// TIA Portal project "PLC_DoAn" (V16)

(* hardware
DEVICE "S71500/ET200MP station_1"  S7-1500 station
   slot 0: "Rail_0"  Rack  6ES7 590-1***0-0AA0
   slot 1: "PLC_1"  CPU 1512C-1 PN  6ES7 512-1CK01-0AB0  V2.8
      slot 3: "CPU display_1"  6ES7591-1AA00-0AA0
      slot 32768: "PROFINET interface_1"  X1
         slot 32769: "Port_1"  X1 P1
         slot 32770: "Port_2"  X1 P2
      slot 34817: "Virtual CP interface port_1"  Virtual CP interface port  Virtual CP interface port
   slot 2: "DQ 16x24VDC/0.5A BA_1"  DQ 16x24VDC/0.5A BA  6ES7 522-1BH10-0AA0  V1.1
DEVICE "PC-System_1"  SIMATIC PC station
   slot 0: "SIMATIC PC station"  Rail  SIMATIC PC-Station  V1.0
      slot 125: "Stationmanager"  Station_Manager  V6.0.4
   slot 1: "HMI_RT_1"  WinCC Unified Scada RT  6AV2 155-xxxxx-xxxx  16.0.0.0
   slot 2: "IE general_1"  IE General  IE_CP  V8.2.0
*)

// ===== PLC "PLC_1"  CPU 1512C-1 PN =====

VAR_GLOBAL   // PLC tag table "Default tag table"
   "Tesst_Alarm" AT %M400.0 : Bool;
   "Reset_Alarm" AT %M400.1 : Bool;
END_VAR

VAR_GLOBAL   // PLC tag table "ControlStep1"
   "highLevelSilo1" AT %M0.0 : Bool;   // sua dia chi
   "lowLevelSilo1" AT %M0.1 : Bool;   // sua dia chi
   "highLevelSilo2" AT %M0.2 : Bool;   // sua dia chi
   "lowLevelSilo2" AT %M0.3 : Bool;   // sua dia chi
   "highLevelSilo3" AT %M0.4 : Bool;   // sua dia chi
   "lowLevelSilo3" AT %M0.5 : Bool;   // sua dia chi
   "highLevelSilo4" AT %M0.6 : Bool;   // sua dia chi
   "lowLevelSilo4" AT %M0.7 : Bool;   // sua dia chi
   "highLevelSilo5" AT %M1.0 : Bool;   // sua dia chi
   "lowLevelSilo5" AT %M1.1 : Bool;   // sua dia chi
   "startPumpSilo1" AT %Q1.2 : Bool;
   "stopPumpSilo1" AT %Q1.3 : Bool;
   "startPumpSilo2" AT %Q1.4 : Bool;
   "stopPumpSilo2" AT %Q1.5 : Bool;
   "startPumpSilo3" AT %Q1.6 : Bool;
   "stopPumpSilo3" AT %Q1.7 : Bool;
   "startPumpSilo4" AT %Q2.0 : Bool;
   "stopPumpSilo4" AT %Q2.1 : Bool;
   "startPumpSilo5" AT %Q2.2 : Bool;
   "stopPumpSilo5" AT %Q2.3 : Bool;
   "errorSilo1" AT %I0.0 : Bool;   // lam alarm
   "errorSilo2" AT %I0.1 : Bool;   // lam alarm
   "errorSilo3" AT %I0.2 : Bool;   // lam alarm
   "errorSilo4" AT %I0.3 : Bool;   // lam alarm
   "errorSilo5" AT %I0.4 : Bool;   // lam alarm
   "levelSilo1" AT %ID92 : Real;
   "levelSilo2" AT %ID96 : Real;
   "levelSilo3" AT %ID88 : Real;
   "levelSilo4" AT %ID112 : Real;
   "levelSilo5" AT %ID116 : Real;
   "speedPumpSilo1" AT %QD92 : Real;
   "speedPumpSilo2" AT %QD96 : Real;
   "speedPumpSilo3" AT %QD108 : Real;
   "speedPumpSilo4" AT %QD112 : Real;
   "speedPumpSilo5" AT %QD116 : Real;
   "fbPumpSupplySilo1" AT %I0.5 : Bool;
   "fbPumpSupplySilo3" AT %I0.7 : Bool;
   "openValveSilo1" AT %Q2.4 : Bool;
   "openValveSilo2" AT %Q2.5 : Bool;
   "openValveSilo3" AT %Q2.6 : Bool;
   "openValveSilo4" AT %Q2.7 : Bool;
   "openValveSilo5" AT %Q3.0 : Bool;
   "closeValveSilo1" AT %Q3.1 : Bool;
   "closeValveSilo2" AT %Q3.2 : Bool;
   "closeValveSilo3" AT %Q3.3 : Bool;
   "closeValveSilo4" AT %Q3.4 : Bool;
   "closeValveSilo5" AT %Q3.5 : Bool;
   "fbOpenValveSilo1" AT %I1.2 : Bool;
   "fbPumpSupplySilo2" AT %I0.6 : Bool;
   "fbPumpSupplySilo4" AT %I1.0 : Bool;
   "fbPumpSupplySilo5" AT %I1.1 : Bool;
   "fbOpenValveSilo2" AT %I1.3 : Bool;
   "fbOpenValveSilo3" AT %I1.4 : Bool;
   "fbOpenValveSilo4" AT %I1.5 : Bool;
   "fbOpenValveSilo5" AT %I1.6 : Bool;
   "fbCloseValveSilo1" AT %I10.0 : Bool;
   "fbCloseValveSilo2" AT %I10.1 : Bool;
   "fbCloseValveSilo3" AT %I10.2 : Bool;
   "fbCloseValveSilo4" AT %I10.3 : Bool;
   "fbCloseValveSilo5" AT %I10.4 : Bool;
END_VAR

VAR_GLOBAL   // PLC tag table "ControlStep2"
   "weightRaw" AT %ID84 : Real;
   "weightRaw1SP" AT %ID124 : Real;
   "weightRaw2SP" AT %ID128 : Real;
   "weightRaw3SP" AT %ID132 : Real;
   "weightSpice" AT %ID104 : Real;
   "weightSpiceSP" AT %ID140 : Real;
   "weightWater" AT %ID100 : Real;
   "weightWaterSP" AT %ID148 : Real;
   "openRaw1ValvePerc" AT %QD120 : Real;
   "openRaw2ValvePerc" AT %QD124 : Real;
   "openRaw3ValvePerc" AT %QD128 : Real;
   "openSpiceValvePerc" AT %QD104 : Real;
   "openWaterValvePerc" AT %QD100 : Real;
   "transferRawDone" AT %I2.0 : Bool;
   "fbOpenValveScaleRaw1" AT %I2.1 : Bool;
   "fbOpenValveScaleRaw2" AT %I2.2 : Bool;
   "fbOpenValveScaleRaw3" AT %I2.3 : Bool;
   "fbOpenValveScaleSpice" AT %I2.4 : Bool;
   "fbOpenValveScaleWater" AT %I2.5 : Bool;
   "fbCloseValveScaleRaw1" AT %I2.6 : Bool;
   "fbCloseValveScaleRaw2" AT %I2.7 : Bool;
   "fbCloseValveScaleRaw3" AT %I3.0 : Bool;
   "fbCloseValveScaleSpice" AT %I3.1 : Bool;
   "fbCloseValveScaleWater" AT %I3.2 : Bool;
   "fbWaterValvePerc" AT %ID108 : Real;
   "fbSpiceValvePerc" AT %ID120 : Real;
END_VAR

VAR_GLOBAL   // PLC tag table "ControlStep3"
   "check" AT %I4.0 : Bool;
   "openValve" AT %Q4.0 : Bool;
END_VAR

VAR_GLOBAL   // PLC tag table "ControlStep4"
   "checkSpice" AT %I6.5 : Bool;
   "checkWater" AT %I6.0 : Bool;
   "openValveSpice" AT %Q6.0 : Bool;
   "openValveWater" AT %Q6.1 : Bool;
   "closeValveSpice" AT %Q6.2 : Bool;
   "closeValveWater" AT %Q6.3 : Bool;
   "fbOpenValveSpice" AT %I6.1 : Bool;
   "fbCloseValveWater" AT %I6.2 : Bool;
   "fbOpenValveWater" AT %I6.3 : Bool;
   "fbCloseValveSpice" AT %I6.4 : Bool;
END_VAR

VAR_GLOBAL   // PLC tag table "ControlStep5"
   "productCheck" AT %I8.0 : Bool;
   "openValveMixer" AT %Q8.0 : Bool;
   "fbOpenValveMIxer" AT %I8.1 : Bool;
END_VAR

TYPE "Alarm_Type"
   STRUCT
      Active : Bool;
      Ack : Bool;
      Latched : Bool;
      Enable : Bool;
   END_STRUCT;
END_TYPE

TYPE "Weight_Alarm_Type"
   STRUCT
      Overweight : "Alarm_Type";
      UnderWeight : "Alarm_Type";
      NoFlow : "Alarm_Type";
      Timeout : "Alarm_Type";
      SensorFault : "Alarm_Type";
      ValveLeak : "Alarm_Type";
   END_STRUCT;
END_TYPE

TYPE "System_Alarm_Type"
   STRUCT
      Water : "Weight_Alarm_Type";
      Additive : "Weight_Alarm_Type";
      Material : "Weight_Alarm_Type";
   END_STRUCT;
END_TYPE

DATA_BLOCK "Recipe"   // DB1
{ S7_Optimized_Access := 'TRUE' }
VERSION : 0.1
   VAR
      maxLevelSilo1 : Real := 0.0;
      minLevelSilo1 : Real := 0.0;
      maxLevelSilo2 : Real := 0.0;
      minLevelSilo2 : Real := 0.0;
      maxLevelSilo3 : Real := 0.0;
      minLevelSilo3 : Real := 0.0;
      maxLevelSilo4 : Real := 0.0;
      minLevelSilo4 : Real := 0.0;
      maxLevelSilo5 : Real := 0.0;
      minLevelSilo5 : Real := 0.0;
      weightOfRaw1 : Real := 0.0;
      weightOfRaw2 : Real := 0.0;
      weightOfRaw3 : Real := 0.0;
      weightOfSpice : Real := 0.0;
      weightOfWater : Real := 0.0;
      errorWeightRaw1 : Real := 2.5;
      errorWeightRaw2 : Real := 2.5;
      errorWeightRaw3 : Real := 2.5;
      errorWeightSpice : Real := 5.0;
      errorWeightWater : Real := 7.0;
      openValvePercMin : Real := 10.0;
   END_VAR
BEGIN
END_DATA_BLOCK

DATA_BLOCK "Control_DB"   // DB2
{ S7_Optimized_Access := 'TRUE' }
VERSION : 0.1
// stored: InstanceOfName Control
"Control"
BEGIN
END_DATA_BLOCK

DATA_BLOCK "Process_DB"   // DB3
{ S7_Optimized_Access := 'TRUE' }
VERSION : 0.1
// stored: InstanceOfName Process
"Process"
BEGIN
END_DATA_BLOCK

DATA_BLOCK "BtnControl"   // DB4
{ S7_Optimized_Access := 'TRUE' }
VERSION : 0.1
   VAR
      start : Bool := false;
      stop : Bool := false;
      auto : Bool := false;
      manu : Bool := false;
      reset : Bool := false;
      pause : Bool := false;
      resume : Bool := false;
      restart : Bool := false;
      hold : Bool := false;
      emerg : Bool := false;
      abort : Bool := false;
      alarm : Bool := false;
      error : Bool := false;
      btn_silo1 : Bool := false;
      btn_silo2 : Bool := false;
      btn_silo3 : Bool := false;
      btn_silo4 : Bool := false;
      btn_silo5 : Bool := false;
      btn_Conveyor : Bool := false;
      btn_scaleRaw1 : Bool := false;
      btn_scaleRaw2 : Bool := false;
      btn_scaleRaw3 : Bool := false;
      btn_scaleSpice : Bool := false;
      btn_scaleWater : Bool := false;
      btn_runGrinder : Bool := false;
      btn_runMixer : Bool := false;
      btn_dischargeSpice : Bool := false;
      btn_dischargeWater : Bool := false;
      btn_dischargeMixer : Bool := false;
      btn_ResetReady : Bool := false;
   END_VAR
BEGIN
END_DATA_BLOCK

DATA_BLOCK "Data"   // DB5
{ S7_Optimized_Access := 'TRUE' }
VERSION : 0.1
   VAR
      state : Int;
      "step" : Int;
      mode : Int;
      set : Bool;
      targetBatches : Int;
      currentBatches : Int;
      silo1Ready : Bool;
      silo2Ready : Bool;
      silo3Ready : Bool;
      silo4Ready : Bool;
      silo5Ready : Bool;
      spiceReady : Bool;
      waterReady : Bool;
      rawReady : Bool;
      grindDone : Bool;
      mixDone : Bool;
      processDone : Bool;
      resetReadyState : Bool;
      enaPumpSilo1 : Bool;
      enaPumpSilo2 : Bool;
      enaPumpSilo3 : Bool;
      enaPumpSilo4 : Bool;
      enaPumpSilo5 : Bool;
      enaScaleRaw1 : Bool;
      enaScaleRaw2 : Bool;
      enaScaleRaw3 : Bool;
      enaScaleSpice : Bool;
      enaScaleWater : Bool;
      runConveyor : Bool;
      runGrinder : Bool;
      runMixer : Bool;
      enaDischargeSpice : Bool;
      enaDischargeWater : Bool;
      enaDischargeMixer : Bool;
      enaNextStep_Raw1 : Bool;
      enaNextStep_Raw2 : Bool;
      weightDoneRaw1 : Bool;
      weightDoneRaw2 : Bool;
      weightDoneRaw3 : Bool;
      enaNextPhase_Grind : Bool;
   END_VAR
BEGIN
END_DATA_BLOCK

DATA_BLOCK "Database_Alarm"   // DB11
{ S7_Optimized_Access := 'FALSE' }
VERSION : 0.1
   VAR
      Alarms : "System_Alarm_Type";
   END_VAR
BEGIN
   // Alarms.Water.UnderWeight : Warning for underweight
   // Alarms.Water.Overweight : Alarm for OverWeight
   // Alarms.Water.NoFlow : Alarm for NoFlow
   // Alarms.Water.Timeout : Warning for Timeout
   // Alarms.Water.ValveLeak : Alarm for ValveLeak
END_DATA_BLOCK

DATA_BLOCK "WeightWater_Alarm_DB"   // DB12
{ S7_Optimized_Access := 'TRUE' }
VERSION : 0.1
// stored: InstanceOfName Weight_Alarm
"Weight_Alarm"
BEGIN
   Ton_NoFlow.PT := T#3S;
   Ton_Timeout.PT := T#30S;
   Ton_Leak.PT := T#2S;
   OverWeight_Limit := 2.0;
   Stability_Range := 0.1;
   T_NoFlow := T#5S;
   T_Timeout := T#5S;
   Leak_Limit := 1.0;
END_DATA_BLOCK

DATA_BLOCK "WeightAdditive_Alarm_DB"   // DB13
{ S7_Optimized_Access := 'TRUE' }
VERSION : 0.1
// stored: InstanceOfName Weight_Alarm
"Weight_Alarm"
BEGIN
   T_NoFlow := T#5S;
   T_Timeout := T#5S;
   OverWeight_Limit := 1.0;
   Stability_Range := 0.1;
   Leak_Limit := 1.0;
END_DATA_BLOCK

// folder: DB

DATA_BLOCK "Phase1_DB"   // DB6
{ S7_Optimized_Access := 'TRUE' }
VERSION : 0.1
// stored: InstanceOfName Phase1
"Phase1"
BEGIN
END_DATA_BLOCK

DATA_BLOCK "Phase2_DB"   // DB7
{ S7_Optimized_Access := 'TRUE' }
VERSION : 0.1
// stored: InstanceOfName Phase2
"Phase2"
BEGIN
END_DATA_BLOCK

DATA_BLOCK "Phase3_DB"   // DB8
{ S7_Optimized_Access := 'TRUE' }
VERSION : 0.1
// stored: InstanceOfName Phase3
"Phase3"
BEGIN
END_DATA_BLOCK

DATA_BLOCK "Phase5_DB"   // DB9
{ S7_Optimized_Access := 'TRUE' }
VERSION : 0.1
// stored: InstanceOfName Phase5
"Phase5"
BEGIN
END_DATA_BLOCK

DATA_BLOCK "Phase4_DB"   // DB10
{ S7_Optimized_Access := 'TRUE' }
VERSION : 0.1
// stored: InstanceOfName Phase4
"Phase4"
BEGIN
END_DATA_BLOCK

DATA_BLOCK "Phase6_DB"   // DB14
{ S7_Optimized_Access := 'TRUE' }
VERSION : 0.1
// stored: InstanceOfName Phase6
"Phase6"
BEGIN
END_DATA_BLOCK

DATA_BLOCK "Phase7_DB"   // DB15
{ S7_Optimized_Access := 'TRUE' }
VERSION : 0.1
// stored: InstanceOfName Phase7
"Phase7"
BEGIN
END_DATA_BLOCK

DATA_BLOCK "Phase8_DB"   // DB16
{ S7_Optimized_Access := 'TRUE' }
VERSION : 0.1
// stored: InstanceOfName Phase8
"Phase8"
BEGIN
END_DATA_BLOCK

DATA_BLOCK "Phase9_DB"   // DB17
{ S7_Optimized_Access := 'TRUE' }
VERSION : 0.1
// stored: InstanceOfName Phase9
"Phase9"
BEGIN
END_DATA_BLOCK

DATA_BLOCK "Phase10_DB"   // DB18
{ S7_Optimized_Access := 'TRUE' }
VERSION : 0.1
// stored: InstanceOfName Phase10
"Phase10"
BEGIN
END_DATA_BLOCK

DATA_BLOCK "Phase11_DB"   // DB19
{ S7_Optimized_Access := 'TRUE' }
VERSION : 0.1
// stored: InstanceOfName Phase11
"Phase11"
BEGIN
END_DATA_BLOCK

DATA_BLOCK "Phase12_DB"   // DB20
{ S7_Optimized_Access := 'TRUE' }
VERSION : 0.1
// stored: InstanceOfName Phase12
"Phase12"
BEGIN
END_DATA_BLOCK

DATA_BLOCK "Phase13_DB"   // DB21
{ S7_Optimized_Access := 'TRUE' }
VERSION : 0.1
// stored: InstanceOfName Phase13
"Phase13"
BEGIN
END_DATA_BLOCK

DATA_BLOCK "Phase14_DB"   // DB22
{ S7_Optimized_Access := 'TRUE' }
VERSION : 0.1
// stored: InstanceOfName Phase14
"Phase14"
BEGIN
END_DATA_BLOCK

DATA_BLOCK "Phase15_DB"   // DB23
{ S7_Optimized_Access := 'TRUE' }
VERSION : 0.1
// stored: InstanceOfName Phase15
"Phase15"
BEGIN
END_DATA_BLOCK

DATA_BLOCK "Phase16_DB"   // DB24
{ S7_Optimized_Access := 'TRUE' }
VERSION : 0.1
// stored: InstanceOfName Phase16
"Phase16"
BEGIN
END_DATA_BLOCK

// folder: (top level)

FUNCTION_BLOCK "Weight_Alarm"   // FB9, SCL
{ S7_Optimized_Access := 'TRUE' }
VERSION : 0.1
   VAR_INPUT
      Weight_SP : Real;
      Weight_PV : Real;
      Valve_Open : Bool;
      Valve_Close : Bool;
      Reset_All : Bool;
      T_NoFlow : Time;
      T_Timeout : Time;
      OverWeight_Limit : Real;
      Stability_Range : Real;
      Leak_Limit : Real;
   END_VAR
   VAR_IN_OUT
      Alarm_Data : "Weight_Alarm_Type";
   END_VAR
   VAR
      Weight_Old : Real;
      Ton_NoFlow : TON_TIME;
      Ton_Timeout : TON_TIME;
      F_Trig_Valve : F_TRIG;
      R_Trig_Close : R_TRIG;
      Weight_At_Close : Real;
      Ton_Leak : TON_TIME;
      Valve_IsOpen : Bool;
      Valve_IsClosed : Bool;
   END_VAR
BEGIN
   // =====================================================
   // 0. QUY ĐỔI TRẠNG THÁI VAN TỪ 2 TÍN HIỆU OPEN/CLOSE
   // =====================================================
   // Chỉ coi là OPEN khi Open=1 và Close=0
   #Valve_IsOpen := #Valve_Open AND NOT #Valve_Close;

   // Chỉ coi là CLOSED khi Close=1 và Open=0
   #Valve_IsClosed := #Valve_Close AND NOT #Valve_Open;

   // Nếu cả 2 cùng 1 hoặc cùng 0 thì không coi là trạng thái hợp lệ
   // Có thể xử lý thêm alarm trạng thái van nếu cần


   // =====================================================
   // 1. XỬ LÝ LOGIC PHÁT HIỆN LỖI (ACTIVE)
   // =====================================================

   // Alarm No Flow:
   // Chỉ giám sát khi van đang MỞ
   #Ton_NoFlow(
               IN := #Alarm_Data.NoFlow.Enable
               AND #Valve_IsOpen
               AND (ABS(#Weight_PV - #Weight_Old) < #Stability_Range),
               PT := #T_NoFlow
   );
   #Alarm_Data.NoFlow.Active := #Ton_NoFlow.Q;


   // Alarm OverWeight:
   // Vẫn kiểm tra bình thường, thường không phụ thuộc trực tiếp trạng thái van
   #Alarm_Data.Overweight.Active :=
   #Alarm_Data.Overweight.Enable
   AND (#Weight_PV > (#Weight_SP + #OverWeight_Limit));


   // Alarm Timeout:
   // Chỉ giám sát khi van đang MỞ
   #Ton_Timeout(
                IN := #Alarm_Data.Timeout.Enable
                AND #Valve_IsOpen,
                PT := #T_Timeout
   );
   #Alarm_Data.Timeout.Active := #Ton_Timeout.Q;


   // =====================================================
   // 2. BẮT THỜI ĐIỂM VAN VỪA ĐÓNG ĐỂ LƯU KHỐI LƯỢNG MỐC
   // =====================================================
   // Dùng cạnh lên của trạng thái CLOSED
   #R_Trig_Close(CLK := #Valve_IsClosed);

   IF #R_Trig_Close.Q THEN
       #Weight_At_Close := #Weight_PV;
   END_IF;


   // =====================================================
   // 3. ALARM RÒ VAN (VALVE LEAK)
   // =====================================================
   // Khi van đang ĐÓNG, nếu cân tiếp tục tăng quá mốc đóng van + Leak_Limit
   // thì sau 2s xác nhận là rò van
   #Ton_Leak(
             IN := #Alarm_Data.ValveLeak.Enable
             AND #Valve_IsClosed
             AND (#Weight_PV > (#Weight_At_Close + #Leak_Limit)),
             PT := T#2s
   );

   #Alarm_Data.ValveLeak.Active := #Ton_Leak.Q;


   // =====================================================
   // 4. XỬ LÝ CHỐT LỖI (LATCHED) VÀ ACK
   // =====================================================

   // -------- NoFlow --------
   IF #Alarm_Data.NoFlow.Active THEN
       #Alarm_Data.NoFlow.Latched := TRUE;
   END_IF;

   IF ((#Reset_All OR #Alarm_Data.NoFlow.Ack) AND NOT #Alarm_Data.NoFlow.Active)
       OR NOT #Alarm_Data.NoFlow.Enable THEN
       #Alarm_Data.NoFlow.Latched := FALSE;
       #Alarm_Data.NoFlow.Ack := FALSE;
   END_IF;


   // -------- Overweight --------
   IF #Alarm_Data.Overweight.Active THEN
       #Alarm_Data.Overweight.Latched := TRUE;
   END_IF;

   IF ((#Reset_All OR #Alarm_Data.Overweight.Ack) AND NOT #Alarm_Data.Overweight.Active)
       OR NOT #Alarm_Data.Overweight.Enable THEN
       #Alarm_Data.Overweight.Latched := FALSE;
       #Alarm_Data.Overweight.Ack := FALSE;
   END_IF;


   // -------- Timeout --------
   IF #Alarm_Data.Timeout.Active THEN
       #Alarm_Data.Timeout.Latched := TRUE;
   END_IF;

   IF ((#Reset_All OR #Alarm_Data.Timeout.Ack) AND NOT #Alarm_Data.Timeout.Active)
       OR NOT #Alarm_Data.Timeout.Enable THEN
       #Alarm_Data.Timeout.Latched := FALSE;
       #Alarm_Data.Timeout.Ack := FALSE;
   END_IF;


   // -------- ValveLeak --------
   IF #Alarm_Data.ValveLeak.Active THEN
       #Alarm_Data.ValveLeak.Latched := TRUE;
   END_IF;

   IF ((#Reset_All OR #Alarm_Data.ValveLeak.Ack) AND NOT #Alarm_Data.ValveLeak.Active)
       OR NOT #Alarm_Data.ValveLeak.Enable THEN
       #Alarm_Data.ValveLeak.Latched := FALSE;
       #Alarm_Data.ValveLeak.Ack := FALSE;
   END_IF;


   // =====================================================
   // 5. CẬP NHẬT GIÁ TRỊ CŨ CHO CHU KỲ SAU
   // =====================================================
   #Weight_Old := #Weight_PV;
END_FUNCTION_BLOCK

FUNCTION_BLOCK "Control"   // FB11, SCL
{ S7_Optimized_Access := 'TRUE' }
VERSION : 0.1
   VAR_INPUT
      start : Bool;
      stop : Bool;
      auto : Bool;
      manu : Bool;
      reset : Bool;
      pause : Bool;
      resume : Bool;
      restart : Bool;
      hold : Bool;
      abort : Bool;
      alarm : Bool;
      error : Bool;
   END_VAR
   VAR_IN_OUT
      mode : Int;
      state : Int;
      "step" : Int;
   END_VAR
BEGIN
   //chon che do hoat dong
   IF #state = 0 THEN
       IF (#auto AND #manu) OR (NOT #auto AND NOT #manu) THEN
           #mode := 0;
       ELSE
           IF #auto THEN
               #mode := 1;
           END_IF;
           IF #manu THEN
               #mode := 2;
           END_IF;
       END_IF;
   END_IF;

   IF #mode <> 0 THEN
       CASE #state OF
           0:
               IF #start THEN
                   #state := 1;
               END_IF;
           1:
               IF #abort THEN
                   #state := 2;
               ELSIF #stop THEN
                   #state := 3;
               ELSIF #pause THEN
                   #state := 4;
               ELSIF #hold THEN
                   #state := 5;
               ELSIF #step = 6 THEN
                   #state := 6;
               END_IF;
           2, 3, 6:
               IF #reset THEN
                   #state := 0;
               END_IF;
           4:
               IF #resume THEN
                   #state := 1;
               END_IF;
           5:
               IF #restart THEN
                   #state := 1;
               END_IF;

       END_CASE;
   END_IF;
END_FUNCTION_BLOCK

FUNCTION_BLOCK "Process"   // FB19, SCL
{ S7_Optimized_Access := 'TRUE' }
VERSION : 0.1
   VAR_INPUT
      state : Int := 0;   // trang thai hoat dong
      mode : Int := 0;   // che do hoat dong, 1: auto, 2: manu
      set : Bool := false;   // tin hieu set cac thong so cai dat
      targetBatches : Int := 0;   // So luong me can lam
      currentBatches : Int := 0;   // So luong me hien tai
      silo1Ready : Bool := false;   // silo 1 da san sang cung cap nguyen lieu
      silo2Ready : Bool := false;   // silo 2 da san sang cung cap nguyen lieu
      silo3Ready : Bool := false;   // silo 3 da san sang cung cap nguyen lieu
      silo4Ready : Bool := false;   // silo 4 da san sang cung cap gia vi
      silo5Ready : Bool := false;   // silo 5 da san sang cung cap nuoc
      spiceReady : Bool := false;   // da can xong gia vi
      waterReady : Bool := false;   // da can xong nuoc
      rawReady : Bool := false;   // da can xong va dua nguyen lieu vao bon nghien
      grindDone : Bool := false;   // da nghien xong nguyen lieu
      mixDone : Bool := false;   // da tron xong nguyen lieu
      processDone : Bool := false;   // xong quy trinh 1 me
      checkProduct : Bool := false;   // ktra sp con trong bon tron ko
      btn_resetReady : Bool := false;   // dkhien reset trang thai ready bang tay (mode manu)
      btn_silo1 : Bool := false;   // dkhien silo bang tay (mode manu)
      btn_silo2 : Bool := false;   // dkhien silo bang tay (mode manu)
      btn_silo3 : Bool := false;   // dkhien silo bang tay (mode manu)
      btn_silo4 : Bool := false;   // dkhien silo bang tay (mode manu)
      btn_silo5 : Bool := false;   // dkhien silo bang tay (mode manu)
      btn_runConveyor : Bool := false;   // dkhien can nguyen lieu bang tay (mode manu)
      btn_scaleRaw1 : Bool := false;   // xa nguyen lieu raw 1 xuong bang tai bang tay (mode manu)
      btn_scaleRaw2 : Bool := false;   // xa nguyen lieu raw 2 xuong bang tai bang tay (mode manu)
      btn_scaleRaw3 : Bool := false;   // xa nguyen lieu raw 3 xuong bang tai bang tay (mode manu)
      btn_scaleSpice : Bool := false;   // dkhien can gia vi bang tay (mode manu)
      btn_scaleWater : Bool := false;   // dkhien can nuoc bang tay (mode manu)
      btn_runGrinder : Bool := false;   // dkhien chay may nghien bang tay (mode manu)
      btn_runMixer : Bool := false;   // dkhien chay may tron bang tay (mode manu)
      btn_DischargeSpice : Bool := false;   // dkhien van gia vi bang tay (mode manu)
      btn_DischargeWater : Bool := false;   // dkhien van nuoc bang tay (mode manu)
      btn_DischargeMixer : Bool := false;   // dkhien van tron bang tay (mode manu)
   END_VAR
   VAR_OUTPUT
      resetReadyState : Bool := false;   // tiep tuc lam me moi -> reset lai cac bien ready
      enaPumpSilo1 : Bool := false;   // cho phep bon 1 bat dau hoat dong
      enaPumpSilo2 : Bool := false;   // cho phep bon 2 bat dau hoat dong
      enaPumpSilo3 : Bool := false;   // cho phep bon 3 bat dau hoat dong
      enaPumpSilo4 : Bool := false;   // cho phep bon 4 bat dau hoat dong
      enaPumpSilo5 : Bool := false;   // cho phep bon 5 bat dau hoat dong
      enaScaleRaw1 : Bool := false;   // cho phep can nguyen lieu 1
      enaScaleRaw2 : Bool := false;   // cho phep can nguyen lieu 2
      enaScaleRaw3 : Bool := false;   // cho phep can nguyen lieu 3
      enaScaleSpice : Bool := false;   // cho phep can gia vi
      enaScaleWater : Bool := false;   // cho phep can nuoc
      runConveyor : Bool := false;   // chay bang tai
      runGrinder : Bool := false;   // chay may nghien
      runMixer : Bool := false;   // chay may tron
      enaDischargeSpice : Bool := false;   // cho phep xa van gia vi vao may tron
      enaDischargeWater : Bool := false;   // cho phep xa van nuoc vao may tron
      enaDischargeMixer : Bool := false;   // cho phep xa hon hop da tron -> hoan thanh 1 batch
   END_VAR
   VAR_IN_OUT
      "step" : Int;
   END_VAR
   VAR
      TP_ResetReadyState : TP_TIME;
   END_VAR
BEGIN
   IF #state = 1 AND #mode = 1 AND #set THEN
       IF #step = 0 AND #currentBatches < #targetBatches THEN
           #step := 1;
       END_IF;

       CASE #step OF
           1:
               IF #silo1Ready AND #silo2Ready AND #silo3Ready AND #silo4Ready AND #silo5Ready THEN
                   #step := 2;
               END_IF;

           2:
               #runConveyor := TRUE;
               #enaScaleRaw1 := TRUE;
               #enaScaleRaw2 := TRUE;
               #enaScaleRaw3 := TRUE;
               #enaScaleWater := TRUE;
               #enaScaleSpice := TRUE;
               IF #rawReady AND #spiceReady AND #waterReady THEN
                   #runConveyor := FALSE;
                   #enaScaleRaw1 := FALSE;
                   #enaScaleRaw2 := FALSE;
                   #enaScaleRaw3 := FALSE;
                   #enaScaleWater := FALSE;
                   #enaScaleSpice := FALSE;
                   #step := 3;
               END_IF;

           3:
               #runGrinder := TRUE;
               IF #grindDone THEN
                   #runGrinder := FALSE;
                   #step := 4;
               END_IF;

           4:
               #runMixer := TRUE;
               #enaDischargeWater := TRUE; //cho phep mo van, mo bao nhieu % tuy thuoc vao phase 14, 15 quyet dinh
               #enaDischargeSpice := TRUE;
               IF #mixDone THEN
                   #runMixer := FALSE;
                   #enaDischargeWater := FALSE;
                   #enaDischargeSpice := FALSE;
                   #step := 5;
               END_IF;

           5:
               #enaDischargeMixer := TRUE;
               IF NOT #checkProduct THEN
                   #currentBatches := #currentBatches + 1;
                   #enaDischargeMixer := FALSE;
                   #step := 0;
               END_IF;
               // reset cac bien ready ve FALSE trong 1s -> chac chan bien nao cung dc reset
               #TP_ResetReadyState.IN := NOT #checkProduct AND #processDone;
               #TP_ResetReadyState.PT := T#1000ms;
               #resetReadyState := #TP_ResetReadyState.Q;
       END_CASE;

   ELSIF #state = 1 AND #mode = 2 AND #set THEN
       #step := 0;
       #resetReadyState := #btn_resetReady;
       //Dk silo
       #enaPumpSilo1 := #btn_silo1;
       #enaPumpSilo2 := #btn_silo2;
       #enaPumpSilo3 := #btn_silo3;
       #enaPumpSilo4 := #btn_silo4;
       #enaPumpSilo5 := #btn_silo5;

       //Dk can va bang tai 
       #runConveyor := #btn_runConveyor;
       #enaScaleRaw1 := #btn_scaleRaw1;
       #enaScaleRaw2 := #btn_scaleRaw2;
       #enaScaleRaw3 := #btn_scaleRaw3;
       #enaScaleWater := #btn_scaleWater;
       #enaScaleSpice := #btn_scaleWater;

       //Dk may nghien va may tron
       #runGrinder := #btn_runGrinder;
       #runMixer := #btn_runMixer;

       //Dong/mo van
       #enaDischargeWater := #btn_DischargeWater;
       #enaDischargeSpice := #btn_DischargeSpice;
       #enaDischargeMixer := #btn_DischargeMixer;
   END_IF;
END_FUNCTION_BLOCK

ORGANIZATION_BLOCK "Alarm"   // OB1, LAD, ProgramCycle
TITLE = "Main Program Sweep (Cycle)"
{ S7_Optimized_Access := 'TRUE' }
VERSION : 0.1
   VAR_INPUT
      Initial_Call : Bool;   // Initial call of this OB
      Remanence : Bool;   // =True, if remanent data are available
   END_VAR
BEGIN

REGION Network 1
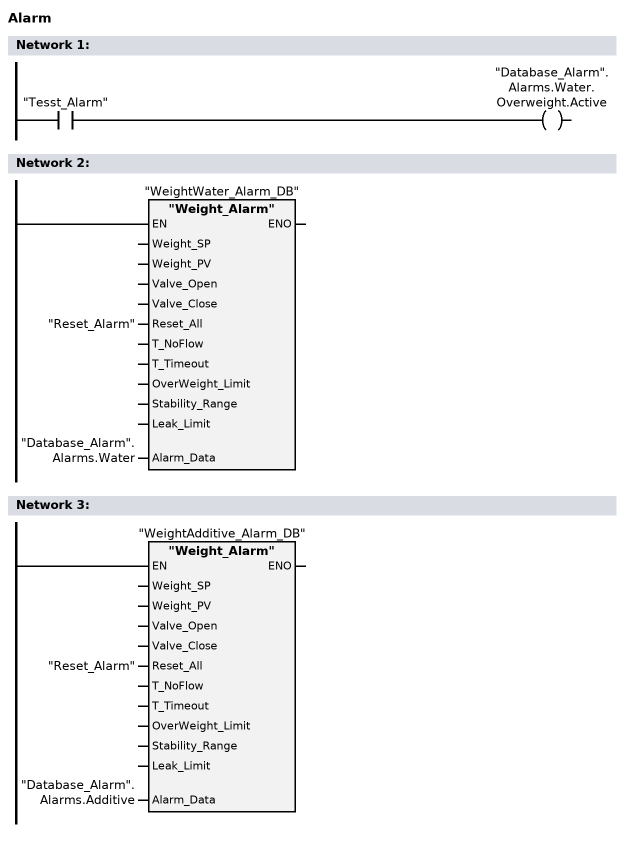
   RUNG wire#powerrail
      Contact( "Tesst_Alarm" )
      Coil( "Database_Alarm".Alarms.Water.Overweight.Active )
   END_RUNG
   // the same network as SCL:
   "Database_Alarm".Alarms.Water.Overweight.Active := "Tesst_Alarm";
END_REGION

REGION Network 2
   RUNG wire#powerrail
      "WeightWater_Alarm_DB"(Weight_SP :=, Weight_PV :=, Valve_Open :=, Valve_Close :=, Reset_All := "Reset_Alarm", T_NoFlow :=, T_Timeout :=, OverWeight_Limit :=, Stability_Range :=, Leak_Limit :=, Alarm_Data := "Database_Alarm".Alarms.Water)
   END_RUNG
   // the same network as SCL:
   "WeightWater_Alarm_DB"(Reset_All := "Reset_Alarm", Alarm_Data := "Database_Alarm".Alarms.Water);   // "Weight_Alarm"
END_REGION

REGION Network 3
   RUNG wire#powerrail
      "WeightAdditive_Alarm_DB"(Weight_SP :=, Weight_PV :=, Valve_Open :=, Valve_Close :=, Reset_All := "Reset_Alarm", T_NoFlow :=, T_Timeout :=, OverWeight_Limit :=, Stability_Range :=, Leak_Limit :=, Alarm_Data := "Database_Alarm".Alarms.Additive)
   END_RUNG
   // the same network as SCL:
   "WeightAdditive_Alarm_DB"(Reset_All := "Reset_Alarm", Alarm_Data := "Database_Alarm".Alarms.Additive);   // "Weight_Alarm"
END_REGION
END_ORGANIZATION_BLOCK

ORGANIZATION_BLOCK "Main"   // OB123, LAD, ProgramCycle
TITLE = "Main Program Sweep (Cycle)"
{ S7_Optimized_Access := 'TRUE' }
VERSION : 0.1
   VAR_INPUT
      Initial_Call : Bool;   // Initial call of this OB
      Remanence : Bool;   // =True, if remanent data are available
   END_VAR
   VAR_TEMP   // added for the SCL form of the ladder/FBD networks
      _w1 : Bool;
      _w2 : Bool;
   END_VAR
BEGIN

REGION Network 1
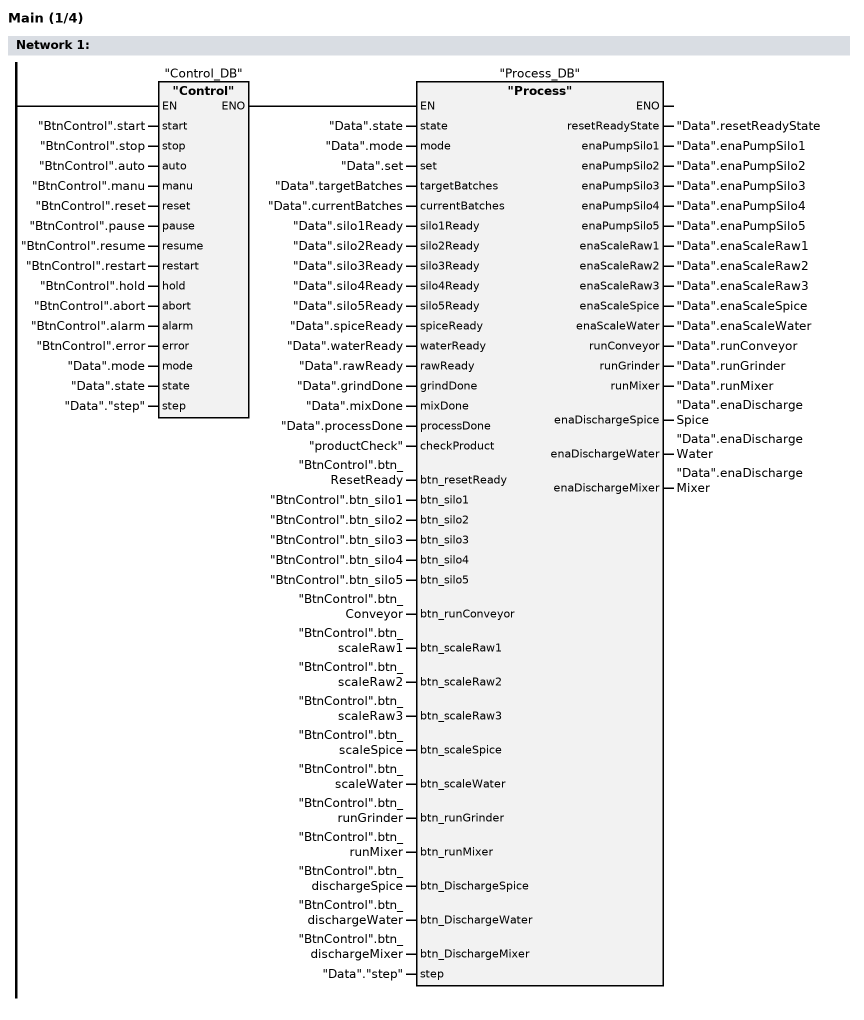
   RUNG wire#powerrail
      "Control_DB"(start := "BtnControl".start, stop := "BtnControl".stop, auto := "BtnControl".auto, manu := "BtnControl".manu, reset := "BtnControl".reset, pause := "BtnControl".pause, resume := "BtnControl".resume, restart := "BtnControl".restart, hold := "BtnControl".hold, abort := "BtnControl".abort, alarm := "BtnControl".alarm, error := "BtnControl".error, mode := "Data".mode, state := "Data".state, "step" := "Data"."step")
      "Process_DB"(state := "Data".state, mode := "Data".mode, set := "Data".set, targetBatches := "Data".targetBatches, currentBatches := "Data".currentBatches, silo1Ready := "Data".silo1Ready, silo2Ready := "Data".silo2Ready, silo3Ready := "Data".silo3Ready, silo4Ready := "Data".silo4Ready, silo5Ready := "Data".silo5Ready, spiceReady := "Data".spiceReady, waterReady := "Data".waterReady, rawReady := "Data".rawReady, grindDone := "Data".grindDone, mixDone := "Data".mixDone, processDone := "Data".processDone, checkProduct := "productCheck", btn_resetReady := "BtnControl".btn_ResetReady, btn_silo1 := "BtnControl".btn_silo1, btn_silo2 := "BtnControl".btn_silo2, btn_silo3 := "BtnControl".btn_silo3, btn_silo4 := "BtnControl".btn_silo4, btn_silo5 := "BtnControl".btn_silo5, btn_runConveyor := "BtnControl".btn_Conveyor, btn_scaleRaw1 := "BtnControl".btn_scaleRaw1, btn_scaleRaw2 := "BtnControl".btn_scaleRaw2, btn_scaleRaw3 := "BtnControl".btn_scaleRaw3, btn_scaleSpice := "BtnControl".btn_scaleSpice, btn_scaleWater := "BtnControl".btn_scaleWater, btn_runGrinder := "BtnControl".btn_runGrinder, btn_runMixer := "BtnControl".btn_runMixer, btn_DischargeSpice := "BtnControl".btn_dischargeSpice, btn_DischargeWater := "BtnControl".btn_dischargeWater, btn_DischargeMixer := "BtnControl".btn_dischargeMixer, "step" := "Data"."step", resetReadyState => "Data".resetReadyState, enaPumpSilo1 => "Data".enaPumpSilo1, enaPumpSilo2 => "Data".enaPumpSilo2, enaPumpSilo3 => "Data".enaPumpSilo3, enaPumpSilo4 => "Data".enaPumpSilo4, enaPumpSilo5 => "Data".enaPumpSilo5, enaScaleRaw1 => "Data".enaScaleRaw1, enaScaleRaw2 => "Data".enaScaleRaw2, enaScaleRaw3 => "Data".enaScaleRaw3, enaScaleSpice => "Data".enaScaleSpice, enaScaleWater => "Data".enaScaleWater, runConveyor => "Data".runConveyor, runGrinder => "Data".runGrinder, runMixer => "Data".runMixer, enaDischargeSpice => "Data".enaDischargeSpice, enaDischargeWater => "Data".enaDischargeWater, enaDischargeMixer => "Data".enaDischargeMixer)
   END_RUNG
   // the same network as SCL:
   "Control_DB"(start := "BtnControl".start,   // "Control"
                stop := "BtnControl".stop,
                auto := "BtnControl".auto,
                manu := "BtnControl".manu,
                reset := "BtnControl".reset,
                pause := "BtnControl".pause,
                resume := "BtnControl".resume,
                restart := "BtnControl".restart,
                hold := "BtnControl".hold,
                abort := "BtnControl".abort,
                alarm := "BtnControl".alarm,
                error := "BtnControl".error,
                mode := "Data".mode,
                state := "Data".state,
                "step" := "Data"."step",
                ENO => #_w1);
   IF #_w1 THEN
       "Process_DB"(state := "Data".state,   // "Process"
                    mode := "Data".mode,
                    set := "Data".set,
                    targetBatches := "Data".targetBatches,
                    currentBatches := "Data".currentBatches,
                    silo1Ready := "Data".silo1Ready,
                    silo2Ready := "Data".silo2Ready,
                    silo3Ready := "Data".silo3Ready,
                    silo4Ready := "Data".silo4Ready,
                    silo5Ready := "Data".silo5Ready,
                    spiceReady := "Data".spiceReady,
                    waterReady := "Data".waterReady,
                    rawReady := "Data".rawReady,
                    grindDone := "Data".grindDone,
                    mixDone := "Data".mixDone,
                    processDone := "Data".processDone,
                    checkProduct := "productCheck",
                    btn_resetReady := "BtnControl".btn_ResetReady,
                    btn_silo1 := "BtnControl".btn_silo1,
                    btn_silo2 := "BtnControl".btn_silo2,
                    btn_silo3 := "BtnControl".btn_silo3,
                    btn_silo4 := "BtnControl".btn_silo4,
                    btn_silo5 := "BtnControl".btn_silo5,
                    btn_runConveyor := "BtnControl".btn_Conveyor,
                    btn_scaleRaw1 := "BtnControl".btn_scaleRaw1,
                    btn_scaleRaw2 := "BtnControl".btn_scaleRaw2,
                    btn_scaleRaw3 := "BtnControl".btn_scaleRaw3,
                    btn_scaleSpice := "BtnControl".btn_scaleSpice,
                    btn_scaleWater := "BtnControl".btn_scaleWater,
                    btn_runGrinder := "BtnControl".btn_runGrinder,
                    btn_runMixer := "BtnControl".btn_runMixer,
                    btn_DischargeSpice := "BtnControl".btn_dischargeSpice,
                    btn_DischargeWater := "BtnControl".btn_dischargeWater,
                    btn_DischargeMixer := "BtnControl".btn_dischargeMixer,
                    "step" := "Data"."step",
                    resetReadyState => "Data".resetReadyState,
                    enaPumpSilo1 => "Data".enaPumpSilo1,
                    enaPumpSilo2 => "Data".enaPumpSilo2,
                    enaPumpSilo3 => "Data".enaPumpSilo3,
                    enaPumpSilo4 => "Data".enaPumpSilo4,
                    enaPumpSilo5 => "Data".enaPumpSilo5,
                    enaScaleRaw1 => "Data".enaScaleRaw1,
                    enaScaleRaw2 => "Data".enaScaleRaw2,
                    enaScaleRaw3 => "Data".enaScaleRaw3,
                    enaScaleSpice => "Data".enaScaleSpice,
                    enaScaleWater => "Data".enaScaleWater,
                    runConveyor => "Data".runConveyor,
                    runGrinder => "Data".runGrinder,
                    runMixer => "Data".runMixer,
                    enaDischargeSpice => "Data".enaDischargeSpice,
                    enaDischargeWater => "Data".enaDischargeWater,
                    enaDischargeMixer => "Data".enaDischargeMixer);
   END_IF;
END_REGION

REGION Network 2: Step 1: Fill silos
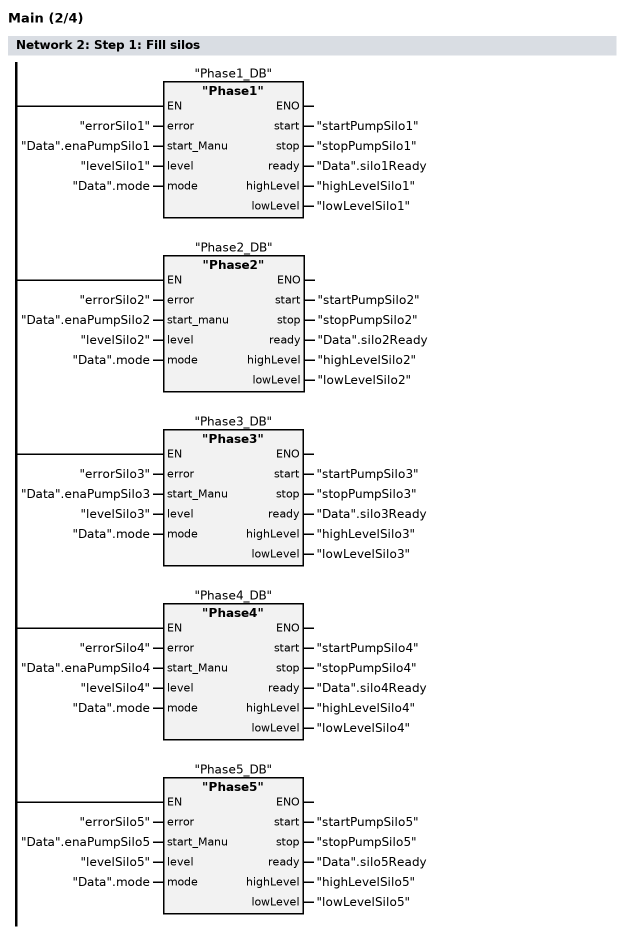
   RUNG wire#powerrail
      "Phase1_DB"(error := "errorSilo1", start_Manu := "Data".enaPumpSilo1, level := "levelSilo1", mode := "Data".mode, start => "startPumpSilo1", stop => "stopPumpSilo1", ready => "Data".silo1Ready, highLevel => "highLevelSilo1", lowLevel => "lowLevelSilo1")
   END_RUNG
   RUNG wire#powerrail
      "Phase2_DB"(error := "errorSilo2", start_manu := "Data".enaPumpSilo2, level := "levelSilo2", mode := "Data".mode, start => "startPumpSilo2", stop => "stopPumpSilo2", ready => "Data".silo2Ready, highLevel => "highLevelSilo2", lowLevel => "lowLevelSilo2")
   END_RUNG
   RUNG wire#powerrail
      "Phase3_DB"(error := "errorSilo3", start_Manu := "Data".enaPumpSilo3, level := "levelSilo3", mode := "Data".mode, start => "startPumpSilo3", stop => "stopPumpSilo3", ready => "Data".silo3Ready, highLevel => "highLevelSilo3", lowLevel => "lowLevelSilo3")
   END_RUNG
   RUNG wire#powerrail
      "Phase4_DB"(error := "errorSilo4", start_Manu := "Data".enaPumpSilo4, level := "levelSilo4", mode := "Data".mode, start => "startPumpSilo4", stop => "stopPumpSilo4", ready => "Data".silo4Ready, highLevel => "highLevelSilo4", lowLevel => "lowLevelSilo4")
   END_RUNG
   RUNG wire#powerrail
      "Phase5_DB"(error := "errorSilo5", start_Manu := "Data".enaPumpSilo5, level := "levelSilo5", mode := "Data".mode, start => "startPumpSilo5", stop => "stopPumpSilo5", ready => "Data".silo5Ready, highLevel => "highLevelSilo5", lowLevel => "lowLevelSilo5")
   END_RUNG
   // the same network as SCL:
   "Phase1_DB"(error := "errorSilo1",   // "Phase1"
               start_Manu := "Data".enaPumpSilo1,
               level := "levelSilo1",
               mode := "Data".mode,
               start => "startPumpSilo1",
               stop => "stopPumpSilo1",
               ready => "Data".silo1Ready,
               highLevel => "highLevelSilo1",
               lowLevel => "lowLevelSilo1");
   "Phase2_DB"(error := "errorSilo2",   // "Phase2"
               start_manu := "Data".enaPumpSilo2,
               level := "levelSilo2",
               mode := "Data".mode,
               start => "startPumpSilo2",
               stop => "stopPumpSilo2",
               ready => "Data".silo2Ready,
               highLevel => "highLevelSilo2",
               lowLevel => "lowLevelSilo2");
   "Phase3_DB"(error := "errorSilo3",   // "Phase3"
               start_Manu := "Data".enaPumpSilo3,
               level := "levelSilo3",
               mode := "Data".mode,
               start => "startPumpSilo3",
               stop => "stopPumpSilo3",
               ready => "Data".silo3Ready,
               highLevel => "highLevelSilo3",
               lowLevel => "lowLevelSilo3");
   "Phase4_DB"(error := "errorSilo4",   // "Phase4"
               start_Manu := "Data".enaPumpSilo4,
               level := "levelSilo4",
               mode := "Data".mode,
               start => "startPumpSilo4",
               stop => "stopPumpSilo4",
               ready => "Data".silo4Ready,
               highLevel => "highLevelSilo4",
               lowLevel => "lowLevelSilo4");
   "Phase5_DB"(error := "errorSilo5",   // "Phase5"
               start_Manu := "Data".enaPumpSilo5,
               level := "levelSilo5",
               mode := "Data".mode,
               start => "startPumpSilo5",
               stop => "stopPumpSilo5",
               ready => "Data".silo5Ready,
               highLevel => "highLevelSilo5",
               lowLevel => "lowLevelSilo5");
END_REGION

REGION Network 3: Step 2: Transfer and scale
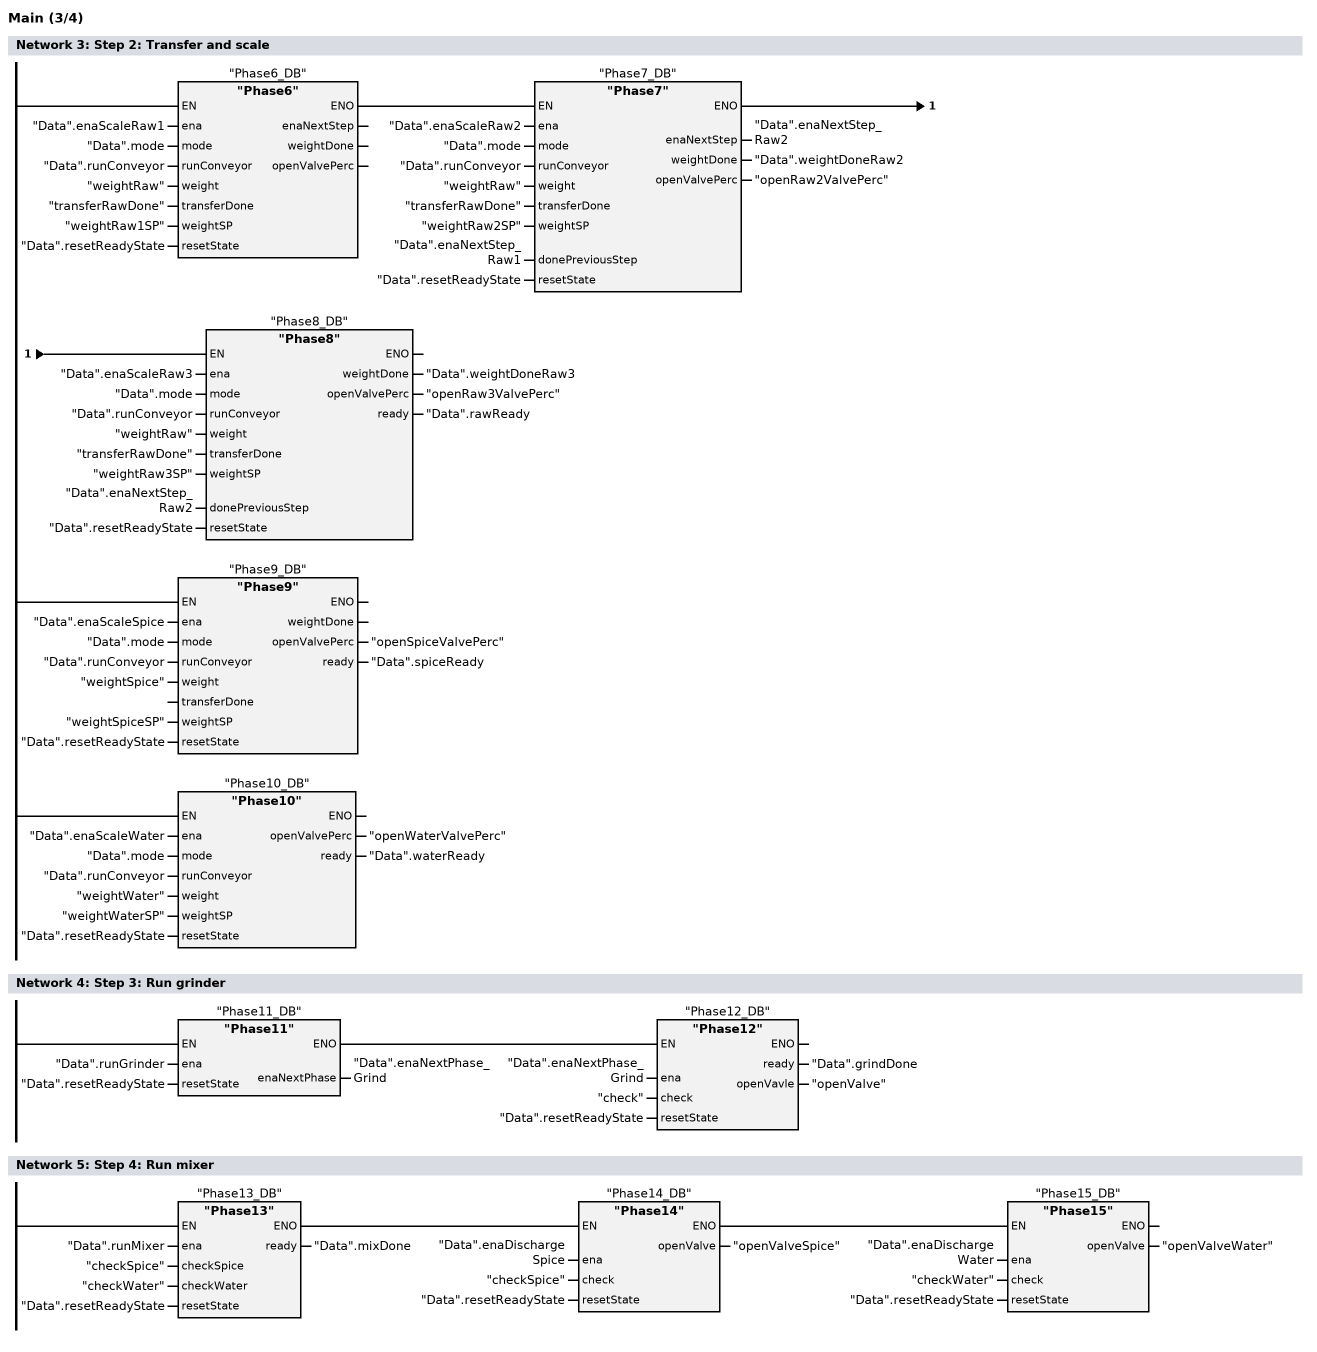
   RUNG wire#powerrail
      "Phase6_DB"(ena := "Data".enaScaleRaw1, mode := "Data".mode, runConveyor := "Data".runConveyor, weight := "weightRaw", transferDone := "transferRawDone", weightSP := "weightRaw1SP", resetState := "Data".resetReadyState, enaNextStep =>, weightDone =>, openValvePerc =>)
      "Phase7_DB"(ena := "Data".enaScaleRaw2, mode := "Data".mode, runConveyor := "Data".runConveyor, weight := "weightRaw", transferDone := "transferRawDone", weightSP := "weightRaw2SP", donePreviousStep := "Data".enaNextStep_Raw1, resetState := "Data".resetReadyState, enaNextStep => "Data".enaNextStep_Raw2, weightDone => "Data".weightDoneRaw2, openValvePerc => "openRaw2ValvePerc")
      "Phase8_DB"(ena := "Data".enaScaleRaw3, mode := "Data".mode, runConveyor := "Data".runConveyor, weight := "weightRaw", transferDone := "transferRawDone", weightSP := "weightRaw3SP", donePreviousStep := "Data".enaNextStep_Raw2, resetState := "Data".resetReadyState, weightDone => "Data".weightDoneRaw3, openValvePerc => "openRaw3ValvePerc", ready => "Data".rawReady)
   END_RUNG
   RUNG wire#powerrail
      "Phase9_DB"(ena := "Data".enaScaleSpice, mode := "Data".mode, runConveyor := "Data".runConveyor, weight := "weightSpice", transferDone :=, weightSP := "weightSpiceSP", resetState := "Data".resetReadyState, weightDone =>, openValvePerc => "openSpiceValvePerc", ready => "Data".spiceReady)
   END_RUNG
   RUNG wire#powerrail
      "Phase10_DB"(ena := "Data".enaScaleWater, mode := "Data".mode, runConveyor := "Data".runConveyor, weight := "weightWater", weightSP := "weightWaterSP", resetState := "Data".resetReadyState, openValvePerc => "openWaterValvePerc", ready => "Data".waterReady)
   END_RUNG
   // the same network as SCL:
   "Phase6_DB"(ena := "Data".enaScaleRaw1,   // "Phase6"
               mode := "Data".mode,
               runConveyor := "Data".runConveyor,
               weight := "weightRaw",
               transferDone := "transferRawDone",
               weightSP := "weightRaw1SP",
               resetState := "Data".resetReadyState,
               ENO => #_w1);
   "Phase7_DB"(EN := #_w1,   // "Phase7"
               ena := "Data".enaScaleRaw2,
               mode := "Data".mode,
               runConveyor := "Data".runConveyor,
               weight := "weightRaw",
               transferDone := "transferRawDone",
               weightSP := "weightRaw2SP",
               donePreviousStep := "Data".enaNextStep_Raw1,
               resetState := "Data".resetReadyState,
               enaNextStep => "Data".enaNextStep_Raw2,
               weightDone => "Data".weightDoneRaw2,
               openValvePerc => "openRaw2ValvePerc",
               ENO => #_w2);
   IF #_w2 THEN
       "Phase8_DB"(ena := "Data".enaScaleRaw3,   // "Phase8"
                   mode := "Data".mode,
                   runConveyor := "Data".runConveyor,
                   weight := "weightRaw",
                   transferDone := "transferRawDone",
                   weightSP := "weightRaw3SP",
                   donePreviousStep := "Data".enaNextStep_Raw2,
                   resetState := "Data".resetReadyState,
                   weightDone => "Data".weightDoneRaw3,
                   openValvePerc => "openRaw3ValvePerc",
                   ready => "Data".rawReady);
   END_IF;
   "Phase9_DB"(ena := "Data".enaScaleSpice,   // "Phase9"
               mode := "Data".mode,
               runConveyor := "Data".runConveyor,
               weight := "weightSpice",
               weightSP := "weightSpiceSP",
               resetState := "Data".resetReadyState,
               openValvePerc => "openSpiceValvePerc",
               ready => "Data".spiceReady);
   "Phase10_DB"(ena := "Data".enaScaleWater,   // "Phase10"
                mode := "Data".mode,
                runConveyor := "Data".runConveyor,
                weight := "weightWater",
                weightSP := "weightWaterSP",
                resetState := "Data".resetReadyState,
                openValvePerc => "openWaterValvePerc",
                ready => "Data".waterReady);
END_REGION

REGION Network 4: Step 3: Run grinder
   RUNG wire#powerrail
      "Phase11_DB"(ena := "Data".runGrinder, resetState := "Data".resetReadyState, enaNextPhase => "Data".enaNextPhase_Grind)
      "Phase12_DB"(ena := "Data".enaNextPhase_Grind, check := "check", resetState := "Data".resetReadyState, ready => "Data".grindDone, openVavle => "openValve")
   END_RUNG
   // the same network as SCL:
   "Phase11_DB"(ena := "Data".runGrinder,   // "Phase11"
                resetState := "Data".resetReadyState,
                enaNextPhase => "Data".enaNextPhase_Grind,
                ENO => #_w1);
   IF #_w1 THEN
       "Phase12_DB"(ena := "Data".enaNextPhase_Grind,   // "Phase12"
                    check := "check",
                    resetState := "Data".resetReadyState,
                    ready => "Data".grindDone,
                    openVavle => "openValve");
   END_IF;
END_REGION

REGION Network 5: Step 4: Run mixer
   RUNG wire#powerrail
      "Phase13_DB"(ena := "Data".runMixer, checkSpice := "checkSpice", checkWater := "checkWater", resetState := "Data".resetReadyState, ready => "Data".mixDone)
      "Phase14_DB"(ena := "Data".enaDischargeSpice, check := "checkSpice", resetState := "Data".resetReadyState, openValve => "openValveSpice")
      "Phase15_DB"(ena := "Data".enaDischargeWater, check := "checkWater", resetState := "Data".resetReadyState, openValve => "openValveWater")
   END_RUNG
   // the same network as SCL:
   "Phase13_DB"(ena := "Data".runMixer,   // "Phase13"
                checkSpice := "checkSpice",
                checkWater := "checkWater",
                resetState := "Data".resetReadyState,
                ready => "Data".mixDone,
                ENO => #_w1);
   "Phase14_DB"(EN := #_w1,   // "Phase14"
                ena := "Data".enaDischargeSpice,
                check := "checkSpice",
                resetState := "Data".resetReadyState,
                openValve => "openValveSpice",
                ENO => #_w2);
   IF #_w2 THEN
       "Phase15_DB"(ena := "Data".enaDischargeWater,   // "Phase15"
                    check := "checkWater",
                    resetState := "Data".resetReadyState,
                    openValve => "openValveWater");
   END_IF;
END_REGION

REGION Network 6: Step 5: Done
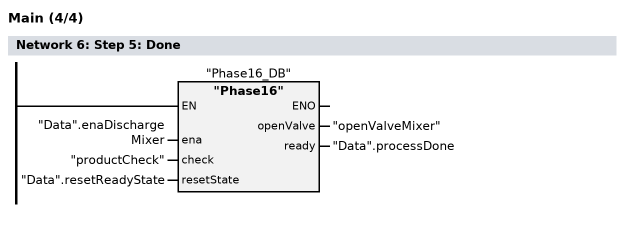
   RUNG wire#powerrail
      "Phase16_DB"(ena := "Data".enaDischargeMixer, check := "productCheck", resetState := "Data".resetReadyState, openValve => "openValveMixer", ready => "Data".processDone)
   END_RUNG
   // the same network as SCL:
   "Phase16_DB"(ena := "Data".enaDischargeMixer,   // "Phase16"
                check := "productCheck",
                resetState := "Data".resetReadyState,
                openValve => "openValveMixer",
                ready => "Data".processDone);
END_REGION
END_ORGANIZATION_BLOCK

// folder: Unit10

FUNCTION_BLOCK "Phase13"   // FB15, SCL
{ S7_Optimized_Access := 'TRUE' }
VERSION : 0.1
   VAR_INPUT
      ena : Bool;
      checkSpice : Bool;
      checkWater : Bool;
      resetState : Bool;
   END_VAR
   VAR_OUTPUT
      ready : Bool;
   END_VAR
   VAR
      TON_RunMixer : TON_TIME;
   END_VAR
   VAR CONSTANT
      "time" : Time := T#10s;
   END_VAR
BEGIN
   #TON_RunMixer.IN := #ena AND #checkSpice AND #checkWater;
   #TON_RunMixer.PT := #time;
   #ready := #TON_RunMixer.Q;
   IF #resetState THEN
       #ready := FALSE;
   END_IF;
END_FUNCTION_BLOCK

FUNCTION_BLOCK "Phase14"   // FB16, SCL
{ S7_Optimized_Access := 'TRUE' }
VERSION : 0.1
   VAR_INPUT
      ena : Bool;
      check : Bool;
      resetState : Bool;
   END_VAR
   VAR_OUTPUT
      openValve : Bool;
   END_VAR
BEGIN
   IF #ena THEN
       #openValve := TRUE;
       IF NOT #check THEN
           #openValve := FALSE;
       END_IF;
   END_IF;
END_FUNCTION_BLOCK

FUNCTION_BLOCK "Phase15"   // FB17, SCL
{ S7_Optimized_Access := 'TRUE' }
VERSION : 0.1
   VAR_INPUT
      ena : Bool;
      check : Bool;
      resetState : Bool;
   END_VAR
   VAR_OUTPUT
      openValve : Bool;
   END_VAR
BEGIN
   IF #ena THEN
       #openValve := TRUE;
       IF NOT #check THEN
           #openValve := FALSE;
       END_IF;
   END_IF;
END_FUNCTION_BLOCK

FUNCTION_BLOCK "Phase16"   // FB18, SCL
{ S7_Optimized_Access := 'TRUE' }
VERSION : 0.1
   VAR_INPUT
      ena : Bool;
      check : Bool;
      resetState : Bool;
   END_VAR
   VAR_OUTPUT
      openValve : Bool;
      ready : Bool;
   END_VAR
BEGIN
   IF #ena THEN
       #openValve := TRUE;
       IF NOT #check THEN
           #openValve := FALSE;
           #ready := TRUE;
       END_IF;
   END_IF;

   IF #resetState THEN
       #ready := FALSE;
   END_IF;
END_FUNCTION_BLOCK

// folder: Unit1_5

FUNCTION_BLOCK "Phase1"   // FB3, SCL
{ S7_Optimized_Access := 'TRUE' }
VERSION : 0.1
   VAR_INPUT
      error : Bool;
      start_Manu : Bool;
      level : Real;
      mode : Int;
   END_VAR
   VAR_OUTPUT
      start : Bool;
      stop : Bool;
      ready : Bool;
      highLevel : Bool;
      lowLevel : Bool;
   END_VAR
BEGIN
   #highLevel := #level >= "Recipe".maxLevelSilo1;
   #lowLevel := #level <= "Recipe".minLevelSilo1;
   #start := #lowLevel;
   #stop := #highLevel OR #error;
   #ready := NOT #highLevel AND NOT #lowLevel;
   IF #mode=2 THEN
       #start := #start_Manu;
   END_IF;
END_FUNCTION_BLOCK

FUNCTION_BLOCK "Phase2"   // FB4, SCL
{ S7_Optimized_Access := 'TRUE' }
VERSION : 0.1
   VAR_INPUT
      error : Bool;
      start_manu : Bool;
      level : Real;
      mode : Int;
   END_VAR
   VAR_OUTPUT
      start : Bool;
      stop : Bool;
      ready : Bool;
      highLevel : Bool;
      lowLevel : Bool;
   END_VAR
BEGIN
   #highLevel := #level >= "Recipe".maxLevelSilo2;
   #lowLevel := #level <= "Recipe".minLevelSilo2;
   #start :=  #lowLevel;
   #stop := #highLevel OR #error;
   #ready := NOT #highLevel AND NOT #lowLevel;
   IF #mode = 2 THEN
       #start := #start_manu;
   END_IF;
END_FUNCTION_BLOCK

FUNCTION_BLOCK "Phase3"   // FB5, SCL
{ S7_Optimized_Access := 'TRUE' }
VERSION : 0.1
   VAR_INPUT
      error : Bool;
      start_Manu : Bool;
      level : Real;
      mode : Int;
   END_VAR
   VAR_OUTPUT
      start : Bool;
      stop : Bool;
      ready : Bool;
      highLevel : Bool;
      lowLevel : Bool;
   END_VAR
BEGIN
   #highLevel := #level >= "Recipe".maxLevelSilo3;
   #lowLevel := #level <= "Recipe".minLevelSilo3;
   #start :=  #lowLevel;
   #stop := #highLevel OR #error;
   #ready := NOT #highLevel AND NOT #lowLevel;
   IF #mode = 2 THEN
       #start := #start_Manu;
   END_IF;
END_FUNCTION_BLOCK

FUNCTION_BLOCK "Phase4"   // FB6, SCL
{ S7_Optimized_Access := 'TRUE' }
VERSION : 0.1
   VAR_INPUT
      error : Bool;
      start_Manu : Bool;
      level : Real;
      mode : Int;
   END_VAR
   VAR_OUTPUT
      start : Bool;
      stop : Bool;
      ready : Bool;
      highLevel : Bool;
      lowLevel : Bool;
   END_VAR
BEGIN
   #highLevel := #level >= "Recipe".maxLevelSilo4;
   #lowLevel := #level <= "Recipe".minLevelSilo4;
   #start :=  #lowLevel;
   #stop := #highLevel OR #error;
   #ready := NOT #highLevel AND NOT #lowLevel;
   IF #mode = 2 THEN
       #start := #start_Manu;
   END_IF;
END_FUNCTION_BLOCK

FUNCTION_BLOCK "Phase5"   // FB7, SCL
{ S7_Optimized_Access := 'TRUE' }
VERSION : 0.1
   VAR_INPUT
      error : Bool;
      start_Manu : Bool;
      level : Real;
      mode : Int;
   END_VAR
   VAR_OUTPUT
      start : Bool;
      stop : Bool;
      ready : Bool;
      highLevel : Bool;
      lowLevel : Bool;
   END_VAR
BEGIN
   #highLevel := #level >= "Recipe".maxLevelSilo5;
   #lowLevel := #level <= "Recipe".minLevelSilo5;
   #start :=  #lowLevel;
   #stop := #highLevel OR #error;
   #ready := NOT #highLevel AND NOT #lowLevel;
   IF #mode = 2 THEN
       #start := #start_Manu;
   END_IF;
END_FUNCTION_BLOCK

// folder: Unit6

FUNCTION_BLOCK "Phase7"   // FB1, SCL
{ S7_Optimized_Access := 'TRUE' }
VERSION : 0.1
   VAR_INPUT
      ena : Bool;
      mode : Int;
      runConveyor : Bool;
      weight : Real;
      transferDone : Bool;
      weightSP : Real;
      donePreviousStep : Bool;
      resetState : Bool;
   END_VAR
   VAR_OUTPUT
      enaNextStep : Bool;
      weightDone : Bool;
      openValvePerc : Real;
   END_VAR
   VAR CONSTANT
      factor : Real := 10.0;
   END_VAR
BEGIN
   IF #ena AND NOT #weightDone AND #mode = 1 AND #donePreviousStep THEN
       IF ABS_REAL(#weight - #weightSP) > "Recipe".errorWeightRaw2 * #factor THEN
           #openValvePerc := 100;
       ELSE
           #openValvePerc := ABS_REAL(#weight - #weightSP) / "Recipe".errorWeightRaw2 * #factor;
           IF #openValvePerc < "Recipe".openValvePercMin THEN
               #openValvePerc := "Recipe".openValvePercMin;
           END_IF;
       END_IF;
   ELSIF #ena AND #mode = 2 THEN
       #openValvePerc := 50;
   ELSE
       #openValvePerc := 0;
   END_IF;

   IF ABS_REAL(#weight - #weightSP) <= "Recipe".errorWeightRaw2 THEN
       #weightDone := TRUE;
   END_IF;

   IF #weightDone AND #transferDone THEN
       #enaNextStep := TRUE;
   END_IF;
   IF #resetState THEN
       #enaNextStep := FALSE;
   END_IF;
END_FUNCTION_BLOCK

FUNCTION_BLOCK "Phase8"   // FB2, SCL
{ S7_Optimized_Access := 'TRUE' }
VERSION : 0.1
   VAR_INPUT
      ena : Bool;
      mode : Int;
      runConveyor : Bool;
      weight : Real;
      transferDone : Bool;
      weightSP : Real;
      donePreviousStep : Bool;
      resetState : Bool;
   END_VAR
   VAR_OUTPUT
      weightDone : Bool;
      openValvePerc : Real;
      ready : Bool;
   END_VAR
   VAR CONSTANT
      factor : Real := 10.0;
   END_VAR
BEGIN
   IF #ena AND NOT #weightDone AND #mode = 1 AND #donePreviousStep THEN
       IF ABS_REAL(#weight - #weightSP) > "Recipe".errorWeightRaw3 * #factor THEN
           #openValvePerc := 100;
       ELSE
           #openValvePerc := ABS_REAL(#weight - #weightSP) / "Recipe".errorWeightRaw3 * #factor;
           IF #openValvePerc < "Recipe".openValvePercMin THEN
               #openValvePerc := "Recipe".openValvePercMin;
           END_IF;
       END_IF;
   ELSIF #ena AND #mode = 2 THEN
       #openValvePerc := 50;
   ELSE
       #openValvePerc := 0;
   END_IF;

   IF ABS_REAL(#weight - #weightSP) <= "Recipe".errorWeightRaw3 THEN
       #weightDone := TRUE;
   END_IF;

   IF #weightDone AND #transferDone THEN
       #ready := TRUE;
   END_IF;
   IF #resetState THEN
       #ready := FALSE;
   END_IF;
END_FUNCTION_BLOCK

FUNCTION_BLOCK "Phase6"   // FB8, SCL
{ S7_Optimized_Access := 'TRUE' }
VERSION : 0.1
   VAR_INPUT
      ena : Bool;
      mode : Int;
      runConveyor : Bool;
      weight : Real;
      transferDone : Bool;
      weightSP : Real;
      resetState : Bool;
   END_VAR
   VAR_OUTPUT
      enaNextStep : Bool;
      weightDone : Bool;
      openValvePerc : Real;
   END_VAR
   VAR CONSTANT
      factor : Real := 10.0;
   END_VAR
BEGIN
   IF #ena AND NOT #weightDone AND #mode = 1 THEN
       IF ABS_REAL(#weight - #weightSP) > "Recipe".errorWeightRaw1 * #factor THEN
           #openValvePerc := 100;
       ELSE
           #openValvePerc := ABS_REAL(#weight - #weightSP) / "Recipe".errorWeightRaw1 * #factor;
           IF #openValvePerc < "Recipe".openValvePercMin THEN
               #openValvePerc := "Recipe".openValvePercMin;
           END_IF;
       END_IF;
   ELSIF #ena AND #mode = 2 THEN
       #openValvePerc := 50;
   ELSE
       #openValvePerc := 0;
   END_IF;

   IF ABS_REAL(#weight - #weightSP) <= "Recipe".errorWeightRaw1 THEN
       #weightDone := TRUE;
   END_IF;

   IF #weightDone AND #transferDone THEN
       #enaNextStep := TRUE;
   END_IF;
   IF #resetState THEN
       #enaNextStep := FALSE;
   END_IF;
END_FUNCTION_BLOCK

// folder: Unit7

FUNCTION_BLOCK "Phase9"   // FB10, SCL
{ S7_Optimized_Access := 'TRUE' }
VERSION : 0.1
   VAR_INPUT
      ena : Bool;
      mode : Int;
      runConveyor : Bool;
      weight : Real;
      transferDone : Bool;
      weightSP : Real;
      resetState : Bool;
   END_VAR
   VAR_OUTPUT
      weightDone : Bool;
      openValvePerc : Real;
      ready : Bool;
   END_VAR
   VAR CONSTANT
      factor : Real := 10.0;
   END_VAR
BEGIN
   IF #ena AND NOT #weightDone AND #mode = 1 THEN
       IF ABS_REAL(#weight - #weightSP) > "Recipe".errorWeightSpice * #factor THEN
           #openValvePerc := 100;
       ELSE
           #openValvePerc := ABS_REAL(#weight - #weightSP) / "Recipe".errorWeightSpice * #factor;
           IF #openValvePerc < "Recipe".openValvePercMin THEN
               #openValvePerc := "Recipe".openValvePercMin;
           END_IF;
       END_IF;
   ELSIF #ena AND #mode = 2 THEN
       #openValvePerc := 50;
   ELSE
       #openValvePerc := 0;
   END_IF;

   IF ABS_REAL(#weight - #weightSP) <= "Recipe".errorWeightSpice THEN
       #weightDone := TRUE;
   END_IF;

   IF #weightDone AND #transferDone THEN
       #ready := TRUE;
   END_IF;
   IF #resetState THEN
       #ready := FALSE;
   END_IF;
END_FUNCTION_BLOCK

// folder: Unit8

FUNCTION_BLOCK "Phase10"   // FB12, SCL
{ S7_Optimized_Access := 'TRUE' }
VERSION : 0.1
   VAR_INPUT
      ena : Bool;
      mode : Int;
      runConveyor : Bool;
      weight : Real;
      weightSP : Real;
      resetState : Bool;
   END_VAR
   VAR_OUTPUT
      openValvePerc : Real;
      ready : Bool;
   END_VAR
   VAR CONSTANT
      factor : Real := 10.0;
   END_VAR
BEGIN
   IF #ena AND NOT #ready AND #mode = 1 THEN
       IF ABS_REAL(#weight - #weightSP) > "Recipe".errorWeightWater * #factor THEN
           #openValvePerc := 100;
       ELSE
           #openValvePerc := ABS_REAL(#weight - #weightSP) / "Recipe".errorWeightWater * #factor;
           IF #openValvePerc < "Recipe".openValvePercMin THEN
               #openValvePerc := "Recipe".openValvePercMin;
           END_IF;
       END_IF;
   ELSIF #ena AND #mode = 2 THEN
       #openValvePerc := 50;
   ELSE
       #openValvePerc := 0;
   END_IF;

   IF ABS_REAL(#weight - #weightSP) <= "Recipe".errorWeightWater THEN
       #ready := TRUE;
   END_IF;

   IF #resetState THEN
       #ready := FALSE;
   END_IF;
END_FUNCTION_BLOCK

// folder: Unit9

FUNCTION_BLOCK "Phase11"   // FB13, SCL
{ S7_Optimized_Access := 'TRUE' }
VERSION : 0.1
   VAR_INPUT
      ena : Bool;
      resetState : Bool;
   END_VAR
   VAR_OUTPUT
      enaNextPhase : Bool;
   END_VAR
   VAR
      TON_RunGrinder : TON_TIME;
   END_VAR
   VAR CONSTANT
      "time" : Time := T#2s;
   END_VAR
BEGIN
   #TON_RunGrinder.IN := #ena;
   #TON_RunGrinder.PT := #time;
   #enaNextPhase := #TON_RunGrinder.Q;

   IF #resetState THEN
       #enaNextPhase := FALSE;
   END_IF;
END_FUNCTION_BLOCK

FUNCTION_BLOCK "Phase12"   // FB14, SCL
{ S7_Optimized_Access := 'TRUE' }
VERSION : 0.1
   VAR_INPUT
      ena : Bool;
      check : Bool;
      resetState : Bool;
   END_VAR
   VAR_OUTPUT
      ready : Bool;
      openVavle : Bool;
   END_VAR
BEGIN
   IF #ena THEN
       #openVavle := TRUE;
       IF #check THEN
           #ready := TRUE;
       END_IF;
   END_IF;
   IF #resetState THEN
       #ready := FALSE;
   END_IF;
END_FUNCTION_BLOCK

(* ===== HMI "HMI_RT_1" =====
connection "HMI_Connection_2": ETHERNET, ILRT_S7_1500_OMS
connection "HMI_Connection_1": ETHERNET, ILRT_S7_1500_OMS

HMI tags "Default tag table"
   "Add_PV_ph14" : Real = PLC Add_PV_ph14 AT %ID34, T1s
   "BltnCLosePump_ph6" : Bool = PLC BltnCLosePump_ph6 AT %I9.1, T1s
   "BltnCLosePump_ph7" : Bool = PLC BltnCLosePump_ph7 AT %I9.5, T1s
   "BltnCLosePump_ph13" : Bool = PLC BltnCLosePump_ph13 AT %I18.1, T1s
   "BltnCLosePump_ph14" : Bool = PLC BltnCLosePump_ph14 AT %I18.5, T1s
   "State" : Int = PLC State AT %MW300, T1s
   "BltnCLoseValve_ph5" : Bool = PLC BltnCLoseValve_ph5 AT %I8.7, T1s
   "BltnCLoseValve_ph6" : Bool = PLC BltnCLoseValve_ph6 AT %I9.3, T1s
   "BltnCLoseValve_ph7" : Bool = PLC BltnCLoseValve_ph7 AT %I9.7, T1s
   "BltnCLoseValve_ph13" : Bool = PLC BltnCLoseValve_ph13 AT %I18.3, T1s
   "BltnCLoseValve_ph14" : Bool = PLC BltnCLoseValve_ph14 AT %I18.7, T1s
   "BltnStopPump_ph4" : Bool = PLC BltnStopPump_ph4 AT %I8.1, T1s
   "BltnStoptPump_ph5" : Bool = PLC BltnStoptPump_ph5 AT %I8.5, T1s
   "BtnOpenPump_ph6" : Bool = PLC BtnOpenPump_ph6 AT %I9.0, T1s
   "BtnOpenPump_ph7" : Bool = PLC BtnOpenPump_ph7 AT %I9.4, T1s
   "BtnOpenPump_ph13" : Bool = PLC BtnOpenPump_ph13 AT %I18.0, T1s
   "BtnOpenPump_ph14" : Bool = PLC BtnOpenPump_ph14 AT %I18.4, T1s
   "BtnOpenValve_ph4" : Bool = PLC BtnOpenValve_ph4 AT %I8.2, T1s
   "BtnOpenValve_ph5" : Bool = PLC BtnOpenValve_ph5 AT %I8.6, T1s
   "BtnOpenValve_ph6" : Bool = PLC BtnOpenValve_ph6 AT %I9.2, T1s
   "BtnOpenValve_ph7" : Bool = PLC BtnOpenValve_ph7 AT %I9.6, T1s
   "BtnOpenValve_ph13" : Bool = PLC BtnOpenValve_ph13 AT %I18.2, T1s
   "BtnOpenValve_ph14" : Bool = PLC BtnOpenValve_ph14 AT %I18.6, T1s
   "BtnStartPump_ph4" : Bool = PLC BtnStartPump_ph4 AT %I8.0, T1s
   "BtnStartPump_ph5" : Bool = PLC BtnStartPump_ph5 AT %I8.4, T1s
   "CloseValve_ph4" : Bool = PLC CloseValve_ph4 AT %Q128.3, T1s
   "CloseValve_ph5" : Bool = PLC CloseValve_ph5 AT %Q128.7, T1s
   "CloseValve_ph6" : Bool = PLC CloseValve_ph6 AT %Q129.1, T1s
   "CloseValve_ph7" : Bool = PLC CloseValve_ph7 AT %Q129.3, T1s
   "CloseValve_ph13" : Bool = PLC CloseValve_ph13 AT %Q129.5, T1s
   "CloseValve_ph14" : Bool = PLC CloseValve_ph14 AT %Q129.7, T1s
   "FB_Close_ValveWeightAdd" : Bool = PLC FB_Close_ValveWeightAdd AT %I5.4, T1s
   "FB_Close_ValveWeightWater" : Bool = PLC FB_Close_ValveWeightWater AT %I5.1, T1s
   "FB_Close_ValveSupplyAdd" : Bool = PLC FB_Close_ValveSupplyAdd AT %I5.3, T1s
   "FB_Close_ValveSupplyWater" : Bool = PLC FB_Close_ValveSupplyWater AT %I5.0, T1s
   "FB_Close_ValveDischargeWeightAdd" : Bool = PLC FB_Close_ValveDischargeWeightAdd AT %I5.5, T1s
   "FB_Close_ValveDischargeWeightWater" : Bool = PLC FB_Close_ValveDischargeWeightWater AT %I5.2, T1s
   "FB_Open_ValveWeightAdd" : Bool = PLC FB_Open_ValveWeightAdd AT %I4.6, T1s
   "FB_Open_ValveWeightWater" : Bool = PLC FB_Open_ValveWeightWater AT %I4.3, T1s
   "FB_Open_ValveSupplyAdd" : Bool = PLC FB_Open_ValveSupplyAdd AT %I4.5, T1s
   "FB_Open_ValveSupplyWater" : Bool = PLC FB_Open_ValveSupplyWater AT %I4.2, T1s
   "FB_Open_ValveDischargeWeightAdd" : Bool = PLC FB_Open_ValveDischargeWeightAdd AT %I4.7, T1s
   "FB_Open_ValveDischargeWeightWater" : Bool = PLC FB_Open_ValveDischargeWeightWater AT %I4.4, T1s
   "FB_PumpSupplyAdd" : Bool = PLC FB_PumpSupplyAdd AT %I4.1, T1s
   "FB_PumpSupplyWater" : Bool = PLC FB_PumpSupplyWater AT %I4.0, T1s
   "HighLevel_ph4" : Bool = PLC HighLevel_ph4 AT %Q3.2, T1s
   "HighLevel_ph5" : Bool = PLC HighLevel_ph5 AT %Q3.3, T1s
   "Level_Additive" : Real = PLC Level_Additive AT %ID14, T1s
   "Level_Water" : Real = PLC Level_Water AT %ID0, T1s
   "LowLevel_ph4" : Bool = PLC LowLevel_ph4 AT %Q3.0, T1s
   "LowLevel_ph5" : Bool = PLC LowLevel_ph5 AT %Q3.1, T1s
   "OpenValve_ph4" : Bool = PLC OpenValve_ph4 AT %Q128.2, T1s
   "OpenValve_ph5" : Bool = PLC OpenValve_ph5 AT %Q128.6, T1s
   "OpenValve_ph6" : Bool = PLC OpenValve_ph6 AT %Q129.0, T1s
   "OpenValve_ph7" : Bool = PLC OpenValve_ph7 AT %Q129.2, T1s
   "OpenValve_ph13" : Bool = PLC OpenValve_ph13 AT %Q129.4, T1s
   "OpenValve_ph14" : Bool = PLC OpenValve_ph14 AT %Q129.6, T1s
   "SpeedPumpAdd" : Real = PLC SpeedPumpAdd AT %QD34, T1s
   "SpeedPumpWater" : Real = PLC SpeedPumpWater AT %QD30, T1s
   "StartPump_ph4" : Bool = PLC StartPump_ph4 AT %Q128.0, T1s
   "StartPump_ph5" : Bool = PLC StartPump_ph5 AT %Q128.4, T1s
   "StopPump_ph4" : Bool = PLC StopPump_ph4 AT %Q128.1, T1s
   "StopPump_ph5" : Bool = PLC StopPump_ph5 AT %Q128.5, T1s
   "ValueValveLevelAdditive" : Real = PLC ValueValveWeightAdditive AT %QD42, T1s
   "ValueValveLevelWater" : Real = PLC ValueValveWeightWater AT %QD38, T1s
   "Water_PV_ph13" : Real = PLC Water_PV_ph13 AT %ID30, T1s
   "Weight_Additive" : Real = PLC Weight_Additive AT %ID26, T1s
   "Weight_Water" : Real = PLC Weight_Water AT %ID22, T1s
   "MixerRunning" : Bool = PLC MixerRunning AT %M200.7, T1s
   "Start" : Bool = PLC Start AT %M100.0, T1s
   "Stop" : Bool = PLC Stop AT %M100.1, T1s
   "Manu" : Bool = PLC Manu AT %M100.3, T1s
   "Auto" : Bool = PLC Auto AT %M100.2, T1s
   "Reset" : Bool = PLC Reset AT %M100.4, T1s
   "Pause" : Bool = PLC Pause AT %M100.5, T1s
   "Hold" : Bool = PLC Hold AT %M101.0, T1s
   "Restart" : Bool = PLC Restart AT %M100.7, T1s
   "Resume" : Bool = PLC Resume AT %M100.6, T1s
   "Emergency" : Bool = PLC Emergency AT %M101.1, T1s
   "Step" : Int = PLC Step AT %MW302, T1s
   "Batch Current" : Real = PLC "Batch Current" AT %MD304, T1s

HMI tags "Alarm_Tag"
   "Alarm_Water_OverWeight" : Bool = PLC Database_Alarm.Alarms.Water.Overweight.Active AT %DB11.DBX0.0, T100ms
   "Alarm_Water_NoFlow" : Bool = PLC Database_Alarm.Alarms.Water.NoFlow.Active AT %DB11.DBX4.0, T100ms
   "Alarm_Water_Timeout" : Bool = PLC Database_Alarm.Alarms.Water.Timeout.Active AT %DB11.DBX6.0, T100ms
   "Alarm_Water_ValveLeak" : Bool = PLC Database_Alarm.Alarms.Water.ValveLeak.Active AT %DB11.DBX10.0, T100ms

discrete alarms
   1: 'Alarm Water OverWeight', class CriticalWithReset, trigger "Alarm_Water_OverWeight" bit 0
   2: 'Alarm Water NoFlow', class Alarm, trigger "Alarm_Water_NoFlow" bit 0
   3: 'Alarm Water Valve Leak', class CriticalWithReset, trigger "Alarm_Water_ValveLeak" bit 0
   4: 'Alarm Water Timeout', class AlarmWithReset, trigger "Alarm_Water_Timeout" bit 0

text list "SystemTextList_ConfigErrorAlarmTextLibrary_1": 1 'NameService configuration error: Implicit deletion - Subelement instance @6%s@ must be deleted explicitly'; 2 'NameService configuration error: Implicit deletion - Alias/Format/Unit instance @6%s@ must be deleted explicitly'

text list "SystemTextList_ConfigErrorAlarmTextLibrary_2": 1 'EvDpManager::cleanupDeletedDatapoint - alert handler config is deleted implicitly for deleted datapoint, @3%s@'; 2 'EvDpManager::cleanupDeletedDatapoint - alert handler config is deleted implicitly but still has overrides, @3%s@'; 3 'EvDpManager::cleanupDeletedDatapoint - default value config is deleted implicitly for deleted datapoint, @3%s@'; 4 'EvDpManager::cleanupDeletedDatapoint - default value config is deleted implicitly but still has overrides, @3%s@'; 5 'EvDpManager::cleanupDeletedDatapoint - initial value config is deleted implicitly for deleted datapoint, @3%s@'; 6 'EvDpManager::cleanupDeletedDatapoint - initial value config is deleted implicitly but still has overrides, @3%s@'; 7 'EvDpManager::cleanupDeletedDatapoint - distribution config is deleted implicitly for deleted datapoint, @3%s@'; 8 'EvDpManager::cleanupDeletedDatapoint - distribution config is deleted implicitly but still has overrides, @3%s@'; 9 'EvDpManager::cleanupDeletedDatapoint - rangeCheck config is deleted implicitly for deleted datapoint, @3%s@'; 10 'EvDpManager::cleanupDeletedDatapoint - rangeCheck config is deleted implicitly but still has overrides, @3%s@'

text list "SystemTextList_ConfigErrorAlarmTextLibrary_3": 1 'DpType has been deleted but there is still a type config defined for the type node, @3%s@'; 2 'DpTypeNode has been deleted in DpType but there is still a type config defined for the element, @3%s@'

text list "SystemTextList_ConfigErrorAlarmTextLibrary_4": 2 'HmiCycle - @6%s@ does not exist'; 3 'HmiAlarm - @6%s@ already exists'; 4 'HmiTag - Address @6%s@ was rejected'; 1 'HmiConnection - @6%s@ does not exist'; 5 'HmiTag - Acquisition mode @6%s@ is not supported by CHROM'; 6 'HmiCycle - @6%s@ deleted, but associated HmiTags exist'; 7 'HmiConnection - @6%s@ deleted, but associated HmiTags exist'; 8 'HmiTag - SelectorTag @6%s@ was rejected'; 9 'HmiTag - SelectorTag @6%s@ has an invalid value'; 0 'Connection could not be established - @6%s@'; 65638 'Connection could not be established - @6%s@'; 65639 'Connection lost - @6%s@'; 65640 'Connection lost on HMI side - @6%s@'; 65641 'Connection lost on PLC side - @6%s@'; 65541 'Connection could not be established - Open timed out - @6%s@'; 65542 'Connection Disturbed - @6%s@'; 65543 'Connection closed on HMI side - HmiConnection @5%s@ is changed'; 65544 'Connection closed on HMI side - Driver attribute is changed - Connection @5%s@'

text list "SystemTextList_ConfigErrorAlarmTextLibrary_5": 1 'HmiConnection - HeartbeatCycle must be lower than HeartbeatResponse'; 2 'HmiConnection - Cyclic Services are configured, but not supported on the target device'; 3 'HmiConnection - Change Driven Read is configured, but not supported on the target device'; 4 'HmiTag - The address @6%s@ does not exist in the PLC'; 5 'HmiTag - The default transformation type for address @6%s@ could not be determined'; 6 'HmiTag - Illegal transformation type.'; 7 'HmiCycle - Cannot be used, transformation is unsupported on HmiCycle'; 4096 'HmiConnection - Address version @6%s@ is not supported yet'; 4097 'HmiConnection - Profibus Addresses are not supported yet'; 4098 'HmiConnection - Softbus Addresses are not supported yet'; 4099 'HmiConnection - Address Type @6%s@ is not supported'; 4100 'HmiConnection - Invalid named connection @6%s@. AccessPoint is ignored'; 4101 'HmiConnection - Routed addresses are not supported. RouteHop @6%s@ won't be used.'; 4102 'HmiConnection - Routed addresses are not supported. RouteNet @6%s@ won't be used.'; 4103 'HmiConnection - Invalid IP address @6%s@'; 4104 'HmiConnection - Invalid named connection @6%s@. Format is supposed to be >VMD</>Connection<'; 4105 'HmiConnection - Invalid named connection @6%s@. VMD too long. At most 24 characters are allowed.'; 4106 'HmiConnection - Invalid named connection @6%s@. Connection too long. At most 32 characters are allowed.'; 4107 'HmiConnection - Rack number @6%s@ is out of range (0..7)'; 4108 'HmiConnection - Invalid named connection @6%s@. Rack is ignored'; 4109 'HmiConnection - Slot number @6%s@ is out of range (1..32)'; 4110 'HmiConnection - Invalid named connection @6%s@. Slot is ignored'; 4111 'Connection could not be established - Maximum number of possible connections (@6%s@) reached'; 4112 'Connection broken - No life sign received in last @6%s@ ms.'; 4113 'Connection could not be established - @5%s@'; 4114 'Connection could not be established - The provided address @6%s@ cannot be used'; 4115 'Connection could not be established - Invalid address @6%s@'; 4116 'Connection could not be established - @5%s@'

text list "SystemTextList_ConfigErrorAlarmTextLibrary_6": 1 'Connection not established - Application instance certificate not configured'; 2 'Connection not established - Server rejected client certificate - OPC UA status code @5%s@'; 3 'Connection not established - Internal certificate store problem - OPC UA status code @5%s@'; 4 'Connection not established - Loading application instance certificate failed - OPC UA status code @5%s@'; 5 'Connection not established - Server has not provided certificate. @5%s@'; 6 'Connection not established - Server certificate validation failed - OPC UA status code @5%s@'; 7 'Connection was closed - Alarm synchronization failed - OPC UA status code @5%s@'; 8 'Connection was closed - Alarm/Event subscription failed due to server operation count limit exceeded'; 9 'Connection was closed - Alarm/Event subscription failed due to server subscription count limit exceeded'; 10 'Connection not established - Server reported license problem - OPC UA status code @5%s@'; 11 'Connection not established - Maximum Number of Server Sessions reached'; 12 'Connection not established - Inconsistent security configuration - @5%s@'; 13 'Connection not established - The provided address @5%s@ cannot be used'; 14 'Connection not established - OPC UA status code @5%s@'; 15 'The connection was lost - OPC UA server was shut down'; 16 'The connection was lost - No life sign received in last @5%s@ milliseconds'; 17 'Connection was closed - OPC UA Server in maintenance'; 18 'Connection not established - Invalid authentication configuration with Authentication Mode - @5%s@'; 19 'Connection not established - User could not be authenticated - OPC UA status code @5%s@'; 20 'Connection not established - Anonymous connection not allowed by server - OPC UA status code @5%s@'; 21 'Connection not established - Certificate problem. Failed to write security relevant file to directory @5%s@'; 22 'Connection not established - Certificate problem. Unexpected file in certificate directory @5%s@ cannot be removed'; 23 'Connection not established - User could not be authenticated - empty userID and password configured'; 24 'Connection not established - Length of configured server certificate exceeded limit. @5%s@'; 25 'Connection not established - Configured @5%s@ has zero length'; 26 'Connection not established - Configured @5%s@ has unexpected format'; 27 'Connection not established - Cannot read endpoints from server. OPC UA status code @5%s@'; 28 'Connection not established - No endpoints found for server. @5%s@'; 29 'Connection not established - Application instance certificate not found.'; 30 'Connection not established - Unexpected format of certificate @5%s@'; 31 'Connection not established - Unexpected format of revocation list @5%s@'; 101 'HmiTag - Provided address @6%s@ does not exist in the server'; 103 'HmiTag - Provided address @6%s@ is not accessible'; 104 'HmiTag - Acquisition Mode not supported for provided address @6%s@'; 201 'HmiAlarm - Provided address @6%s@ does not exist in the server'; 202 'HmiAlarm - Provided address @6%s@ cannot be used because the area filter provided is not an OPC UA event notifier'; 203 'HmiAlarm - Provided address @6%s@ cannot be used because the area filter provided does not exist in the server'; 204 'HmiAlarm - Provided address @6%s@ cannot be used because it is not an OPC UA event type'; 205 'HmiAlarm - Provided address @6%s@ cannot be used because the OPC UA condition type is not supported'; 206 'HmiAlarm - Provided address @6%s@ cannot be used because the event type provided does not exist in the server'; 207 'HmiAlarm - Acquisition Mode value not supported for provided address @6%s@'; 301 'Provided address @6%s@ cannot be used because it is missing version'; 302 'Provided address @6%s@ cannot be used because it contains invalid version'; 303 'Provided address @6%s@ cannot be used because it has invalid count of separators '$''; 304 'Provided address @6%s@ cannot be used because the address kind is invalid'; 305 'Unsupported version @6%s@ of Address'; 401 'Unexpected OPC UA Server response: @6%s@'

text list "SystemTextList_ConfigErrorAlarmTextLibrary_7": 1 'AlarmAnnunciator - Invalid condition string for annunciator @6%s@'; 2 'AlarmAnnunciator - Invalid state tag and bit for annunciator @6%s@'; 3 'AlarmAnnunciator - Invalid silence control tag and bit for annunciator @6%s@'

text list "SystemTextList_ConfigErrorAlarmTextLibrary_8": 1 'TagLogging configuration error: implicit deletion - LoggingTag instance @6%s@ should be deleted but has overrides'

text list "SystemTextList_ConfigErrorAlarmTextLibrary_9": 1 ''; 2 'Restart of the runtime is required!'; 3 'Eject and insert of correct media is required!'

text list "SystemTextList_S7PlusAlarmTextListCollection_1": 4096 'Connection lost on PLC side - @5%s@'; 4097 'Connection lost on HMI side - @5%s@'; 4098 'Maximum number of connections exceeded - @5%s@'; 4099 'Out of resources on PLC - @5%s@'; 4100 'Legitimation failed, invalid or missing password - @5%s@'; 4101 'Open request failed - @5%s@'; 4102 'Cannot connect to PLC - @5%s@'; 4103 'Open request could not be sent'

text list "State": 0 'Idle'; 1 'Running'

graphic list "Pump": 0 'Graphic_116'; 1 'Graphic_117'

graphic list "Valve1": 0 'Graphic_119'; 1 'Graphic_118'

graphic list "Motor": 0 'Graphic_2'; 1 'Graphic_8'
*)